# B&R Automation Studio project 305841_E00002_AM_0 (part 3)

#### GAMath.fun - Exported functions and function blocks
```iecst
(********************************************************************
 * COPYRIGHT -- General Atomics
 ********************************************************************
 * Library: GAMath
 * File: GAMathj.fun
 * Author: J Sheeron
 ********************************************************************
 * Functions and function blocks of library GAMath
 ********************************************************************)

FUNCTION_BLOCK fbCalcTrapMoveTime
  VAR_INPUT
    _I_Vel0 : REAL := 0.0; (* units/sec starting velocity *)
    _I_VelMove : REAL; (* units/sec desired move velocity*)
    _I_Accel : REAL; (* untis/sec^2 *)
    _I_Decel : REAL; (* untis/sec^2 *)
    _I_Dist : LREAL; (* units, LREAL to be compatible with motion system *)
  END_VAR

  VAR_OUTPUT
    _O_MoveTime : TIME; (* how long will the move take as a TIME type *)
    _O_MoveTimeMsec : DINT; (* mSec, how long the move will take *)
    _O_VelReached : REAL; (* units/sec. Velocity reached will be <= VelMove for triangular profiles, dist < Dcheck *)
    _O_Dcheck : LREAL; (* units. Distances > than this have a trapazoidal shape and VelReached = VelMove *)
  END_VAR

  VAR
    v0 : REAL; (* internal copy of input *)
    vMove : REAL; (* internal copy of input *)
    accel : REAL; (* internal copy of input *)
    decel : REAL; (* internal copy of input *)
    dist : LREAL; (* internal copy of input *)
    tval1  : LREAL; (* temporary value *)
    tval2  : LREAL; (* temporary value *)
    tval3  : LREAL; (* temporary value *)
    tval4  : LREAL; (* temporary value *)
    tval5  : LREAL; (* temporary value *)
    seconds : LREAL; (* temporary value *)
  END_VAR
END_FUNCTION_BLOCK

FUNCTION fctAziDiff : LREAL (* Return the angle between pos A and pos B (A-B). Returns +/- 180 deg. +: Pos A ahead of B, -: Pos A behind B *)
  (*
  Result is +/- 180 degrees
  Positive value: A is ahead of B.
  Negative value: A is behind B.
  Account for 360 deg rollover. *)
  VAR_INPUT
    _I_PosA : LREAL;
    _I_PosB : LREAL;
  END_VAR

  VAR
    angle : LREAL;
  END_VAR
END_FUNCTION

FUNCTION fctLRCeiling : LREAL (* LREAL Ceiling -- Return the smallest whole number not less than value *)
  VAR_INPUT
    _I_Val : LREAL;
  END_VAR

  VAR
    val1 : LREAL;
    rem : LREAL;
  END_VAR
END_FUNCTION

FUNCTION fctLRFloor : LREAL (* LREAL floor -- Return the largest whole number not greater than value *)
  VAR_INPUT
    _I_Val : LREAL;
  END_VAR

  VAR
    val1 : LREAL;
  END_VAR
END_FUNCTION

FUNCTION fctLRFract : LREAL (* LREAL fractional -- Return the fractional part of a value *)
  VAR_INPUT
    _I_Val : LREAL;
  END_VAR

  VAR
    val1 : LREAL;
  END_VAR
END_FUNCTION

FUNCTION fctLRMod : LREAL (* LREAL MOD -- Return the remainder of Dividend MOD Divisor *)
  VAR_INPUT
    _I_Dividend : LREAL;
    _I_Divisor : LREAL;
  END_VAR

  VAR
    val1 : LREAL;
    rem : LREAL;
  END_VAR
END_FUNCTION

FUNCTION fctRound1 : REAL (* Return the source value (real) rounded to 1 decimal place *)
  VAR_INPUT
    _I_src : LREAL; (* REAL value to be rounded *)
  END_VAR
  VAR
    dintTemp : DINT; (* temp value *)
  END_VAR
END_FUNCTION

FUNCTION fctRound2 : REAL (* Return the source value (real) rounded to 2 decimal places *)
  VAR_INPUT
    _I_src : LREAL; (* REAL value to be rounded *)
  END_VAR
  VAR
    dintTemp : DINT; (* temp value *)
  END_VAR
END_FUNCTION

FUNCTION fctRound3 : REAL (* Return the source value (real) rounded to 2 decimal places *)
  VAR_INPUT
    _I_src : LREAL; (* REAL value to be rounded *)
  END_VAR
  VAR
    dintTemp : DINT; (* temp value *)
  END_VAR
END_FUNCTION

FUNCTION fctLRound1 : LREAL (* Return the source value (LREAL) rounded to 1 decimal place *)
  VAR_INPUT
    _I_src : LREAL; (* REAL value to be rounded *)
  END_VAR
  VAR
    dintTemp : DINT; (* temp value *)
  END_VAR
END_FUNCTION

FUNCTION fctLRound2 : LREAL (* Return the source value (LREAL) rounded to 2 decimal places *)
  VAR_INPUT
    _I_src : LREAL; (* REAL value to be rounded *)
  END_VAR
  VAR
    dintTemp : DINT; (* temp value *)
  END_VAR
END_FUNCTION

FUNCTION fctLRound3 : LREAL (* Return the source value (LREAL) rounded to 2 decimal places *)
  VAR_INPUT
    _I_src : LREAL; (* REAL value to be rounded *)
  END_VAR
  VAR
    dintTemp : DINT; (* temp value *)
  END_VAR
END_FUNCTION
```

#### GAMath.st - Implementation code
```iecst
(********************************************************************
 * COPYRIGHT -- General Atomics
 ********************************************************************
 * Library: GAMath
 * File: GAMathj.st
 * Author: J Sheeron
 ********************************************************************
 * Functions and function blocks of library GAMath
 ********************************************************************)
// Estimate time needed to make a trapazoidal move
FUNCTION_BLOCK fbCalcTrapMoveTime

  // Useful motion formulas:
  //    V^2 = V0^2 + (2 * acc * dist)  OR  dist = (V^2 - V0^2) / 2acc (1)
  //    V = V0 + (acc * t)  OR  t = (V - V0) / acc                    (2)
  //    Dist = (V0*t) + (1/2 * acc * t^2)                             (3)

  // **** First, return zeros on invalid inputs.
  // Assume distance, and accel and decel cannot be zero.
  // Assume V - V0 cannot be zero
  IF _I_VelMove = 0.0 OR (_I_VelMove = _I_Vel0) OR _I_Accel = 0.0 OR _I_Decel = 0.0 OR _I_Dist = 0.0 THEN
    _O_MoveTime := T#0ms;
    _O_VelReached := 0.0;
    _O_Dcheck := 0.0;
    RETURN;
  END_IF;

  // **** Condition inputs.
  // Force accel, decel and distance to be positive.
  // Force VelMove > V0, swapping them if necessary.
  // IMPROVEMENT: Perhaps it can be made so that negative accel, decel, distance, and velocity inputs
  // are handled gracrfully. Not needed now, so leave this for later if there is time/need.
  v0 := ABS(_I_Vel0);
  vMove := ABS(_I_VelMove);
  // swap V0 and VMove if needed such that v0 < vMove
  IF v0 > vMove THEN
    v0 := ABS(_I_VelMove);
    vMove := ABS(_I_Vel0);
  END_IF;
  accel := ABS(_I_Accel);
  decel := ABS(_I_Decel);
  dist := ABS(_I_Dist);

  // **** Now figure out the move profile.
  // If the requested distance is less than or equal the check distance Dcheck,
  // the move profile is a triangle, and the move velocity will not be reached,
  // or may be reached, but not sustained.

  // If the requested distance is greater than the check distance, then the
  // move profile is trapazoidal, and the velocity will flat top at the move velocity.

  // Calculate the check distance Dcheck
  tval1 := vMove**2 - v0**2;
  tval2 := tval1 / (2 * accel); // dist accel (V^2 - V0^2) / (2*accel) (1)
  tval3 := tval1 / (2 * decel); // dist decel
  _O_Dcheck := tval2 + tval3; // Return the distance check for informational purposes.

  IF dist <= _O_Dcheck THEN
    // ** Triangular profiles
    // Profile is an accel segment and decel segemnt that meet at a point (no flat top at the MOVE velocity).
    // We need to know what velocity is reached. ** The area of the triangle is the distance traveled**,
    // and we know the accel time or distance + the decel time or distance = total time or distance, but we
    // need to know how long or how far the accel or decel component is.
    // Dist = 1/2 * acc * t^2 (3) above, so distance (area) varies linearly and inversely with acc. Furthermore,
    // we know the ratio of accel to decel, so we should be able to figure out the ratio of the distances (areas).
    // Daccel = (1 / Ratio accel:decel) * Ddecel ==> Daccel = (decel/accel) * Ddecel  OR  Ddecel = (accel / decel) * Daccel  (4)
    // Dtotal = Taccel + Tdecel. Substituing in (4) ==> Dtotal = Daccel + (accel/decel) * Daccel ==>
    // Dtotal = Daccel(1 + accel/decel) OR Daccel = Dtotal / (1 + (accel / decel))
    // The area of the acceleration portion is the trialgle with a base with a length of time Tacc, and this varies with the total time
    // by the same ratio of the accel/decel because the area of the triangle varies linearly with the length of the base
    // Taccel = (1 / Ratio accel:decel) * Tdecel ==> Taccel = (decel/accel) * Tdecel OR Tdecel = (accel / decel) * Taccel    (5)
    // Ttotal = Taccel + Tdecel. Substituing in (4) ==> Ttotal = Taccel + (accel/decel) * Taccel ==>
    // Ttotal = Taccel(1 + accel/decel) OR Taccel = Ttotal / (1 + (accel / decel))
    // So putting this all together:
    // 1) Distance traveled = area of the triangle
    // 2) The length of the base of the triangle is the total time
    // 3) Aaccel = Daccel = Dtotal / (1 + (accel / decel)
    // Then it follows that:
    // 4) V = SQRT(V0^2 + (2 * accel * Daccel))             (1)
    // 5) Ttotal = ((V - V0) / accel) + ((V - V0) / decel)  (2)
    tval1 := dist / (1 + (accel / decel));  // Daccel
    _O_VelReached := SQRT(v0**2 + (2.0 * accel * tval1)); // V = SQRT(V0^2 + (2 * acc * dist))
    tval1 := _O_VelReached - v0;
    seconds :=  (tval1 / accel) + (tval1 / decel); // Move time as a float, in seconds. t = ((V - V0) / accel) + ((V - V0) / decel)
  ELSE
    // trapazoidal profiles -- profile is an accel segment a decel segemnt,
    // and a constant velocity segment in between at the move velocity.
    // Total move time is Taccel + Tconstant + Tdecel.
    // Velocity reached = move velocity.
    _O_VelReached := vMove;

    // 1) Calculate the time it takes to accelerate to Vmove
    // Taccel = (V - V0) / accel   (2)
    // 2) Calculate the distance traveled during the acceleration segment
    // Daccel = 1/2 * accel * t^2  (3)
    // 3) Similarly calcuate Tdecel and Ddecel
    // 4) Dconstant = Dmove - (Daccel + Ddecel) Total distance less distance for accel & decel
    // 5) Tconstant = Dconstant / Vmove
    // 6) Calculate Total move time: Tmove = Taccel + Tconstant + Tdecel

    // Calc accel and decel times
    tval1 := vMove - v0;
    tval2 := tval1 / accel; // Taccel = (V - V0) / accel  (2)
    tval3 := tval1 / decel; // Tdecel

    // Calc accel and decel distances
    tval4 := (v0 * tval2) + (0.5 * accel * (tval2**2)); // Daccel = V0*t + (1/2 * accel * t^2)  (3)
    tval5 := (v0 * tval3) + (0.5 * decel * (tval3**2)); // Ddecel

    // Calc constant velocity distance: Dtotal - (Daccel + Ddecel)
    tval1 := dist - (tval4 + tval5); // Dconstant

    // Calc constant velocity time: Tconstant = Dconstant / VMove
    tval4 := tval1 / vMove; // Tconstant

    // Calc Total seconds = Tmove = Taccel + Tconstant + Tdecel
    seconds := tval2 + tval4 + tval3;
  END_IF;

  // Time calculations is:
  // 1) Converted from seconds to mSec (conversion to time expects mSecs)
  // 2) Converted from LREAL to DINT, and then returned for convenience
  // 3) Converted to a TIME and returned.
  _O_MoveTimeMsec := LREAL_TO_DINT(1000 * seconds);
  _O_MoveTime := DINT_TO_TIME(_O_MoveTimeMsec);
END_FUNCTION_BLOCK

// Return the angle between pos A and pos B (A-B). Returns +/- 180 deg. +: Pos A ahead of B, -: Pos A behind B
FUNCTION fctAziDiff
  // Positive value: A is ahead of B,
  // Negative value: A is behind B.
  // Accounts for 360 degree rollover

  angle := _I_PosA - _I_PosB;
  // Deal with 360 deg rollover and normalize result to +/- 180 deg
  // Subtract target from position.
  // If the result < -180, add 360.
  // If the result > 180, subtract 360.
  IF angle < -180.0 THEN
    angle:= angle + 360.0;
  ELSIF angle > 180.0THEN
    angle := angle - 360.0;
  END_IF;
  fctAziDiff := angle;
END_FUNCTION

// LREAL Ceiling -- Return the smallest whole number not less than value
FUNCTION fctLRCeiling
  val1 := TRUNC(_I_Val);
  rem := _I_Val - val1; // the remainder portion
  IF rem > 0 THEN
    // non-zero remainder. Round up
    fctLRCeiling := val1 + 1.0;
  ELSE
    // no remainder -- must already be a whole number
    fctLRCeiling := val1;
  END_IF;
END_FUNCTION

// LREAL Floor -- Return the largest whole number as a LREAL not greater than value
FUNCTION fctLRFloor
  val1 := TRUNC(_I_Val);  // Trunc returns an integer, but it is put into a LREAL
  fctLRFloor := val1;
END_FUNCTION

// LREAL Fract -- Return the fractional part of a value
FUNCTION fctLRFract
  val1 := TRUNC(_I_Val);
  fctLRFract := _I_Val - val1; // the remainder portion
END_FUNCTION

// MOD LREAL Return the remainder of Dividend MOD Divisor
FUNCTION fctLRMod
  val1 := _I_Dividend / _I_Divisor;
  rem := val1 - TRUNC(val1); // the remainder portion
  fctLRMod := rem * _I_Divisor; // remainder * divisor = mod
END_FUNCTION

// Return the source value (real) rounded to 1 decimal place
FUNCTION fctRound1
  dintTemp:= LREAL_TO_DINT(_I_src * 10.0);
  fctRound1:= DINT_TO_REAL(dintTemp) / 10.0;
END_FUNCTION

// Return the source value (real) rounded to 2 decimal places
FUNCTION fctRound2
  // On SG4 systems the REAL_TO_DINT function rounds.
  // Beware that on SG3 systems, it truncates.
  dintTemp:= LREAL_TO_DINT(_I_src * 100.0);
  fctRound2:= DINT_TO_REAL(dintTemp) / 100.0;
END_FUNCTION

// Return the source value (real) rounded to 3 decimal places
FUNCTION fctRound3
  // On SG4 systems the REAL_TO_DINT function rounds.
  // Beware that on SG3 systems, it truncates.
  dintTemp:= LREAL_TO_DINT(_I_src * 1000.0);
  fctRound3:= DINT_TO_REAL(dintTemp) / 1000.0;
END_FUNCTION

// Return the source value (LREAL) rounded to 1 decimal place
FUNCTION fctLRound1
  dintTemp:= LREAL_TO_DINT(_I_src * 10.0);
  fctLRound1:= DINT_TO_LREAL(dintTemp) / 10.0;
END_FUNCTION

// Return the source value (LREAL) rounded to 2 decimal places
FUNCTION fctLRound2
  // On SG4 systems the REAL_TO_DINT function rounds.
  // Beware that on SG3 systems, it truncates.
  dintTemp:= LREAL_TO_DINT(_I_src * 100.0);
  fctLRound2:= DINT_TO_LREAL(dintTemp) / 100.0;
END_FUNCTION

// Return the source value (LREAL) rounded to 3 decimal places
FUNCTION fctLRound3
  // On SG4 systems the REAL_TO_DINT function rounds.
  // Beware that on SG3 systems, it truncates.
  dintTemp:= LREAL_TO_DINT(_I_src * 1000.0);
  fctLRound3:= DINT_TO_LREAL(dintTemp) / 1000.0;
END_FUNCTION
```

### Logic.typ
```iecst
TYPE
  eAXIS_DESIGNATION :
    ( (* Physical Axes *)
    AD_UNKNOWN := 0,
    AD_SPINDLE := 1,
    AD_OUTER_ECCENTRIC := 2,
    AD_INNER_ECCENTRIC := 3,
    AD_Z := 4,
    (* Other axes *)
    AD_X := 5, (* depth *)
    AD_Y := 6, (* used ? *)
    (* virtual axis *)
    AD_HANDWHEEL := 7,
    (* VFD axis *)
    AD_CF_VFD := 8
  ) := AD_UNKNOWN;

  (* Machine specific HMI axis requests. Intended to have one of these structures per axis. *)
  sHmiAxisReqs : STRUCT
    (* Boolean requests in this section. *)
    (* (none *)
    (* numerical requests *)
    (* (none *)
    (* hmi move type and direction selection related *)
    absMoveEnable : BOOL := TRUE; (* allow move type selection by default *)
    relMoveEnable : BOOL := TRUE;
    velMoveEnable : BOOL := TRUE;
    directionPosEnable : BOOL := TRUE; (* allow direction selection by default *)
    directionNegEnable : BOOL := TRUE;
    directionShortestEnable : BOOL := TRUE;
    moveDistanceEnable : BOOL := TRUE; (* enable params by default *)
    movePositionEnable : BOOL := TRUE;
    gearInEnable : BOOL := FALSE; (* coodinated axis gear in enabled *)
    shiftEnable : BOOL := FALSE; (* coordinated axis gear offset or phase shift  enabled *)
    camInEnable : BOOL := FALSE; (* coordinated axis cam in enabled *)
    disengageEnable : BOOL := FALSE; (* coordinated axis cam in enabled *)
    moveDesignation: DINT := -1; (* per hmi. 0: Abs, 1: Rel, 2:Vel or Jog, -1 is no selection. See fctDecodeHmiMoveType *)
    direction: DINT := -1; (* per hmi. 0: pos, 1: neg, 2: shortest, -1 is no selection. See fctDecodeHmiDirection *)
    (* axis designation. Two different data types for convenience. *)
    axisNo : USINT := 0; (* default to initial so setting a value can be detected. USINT for easy use in loops *)
    axisDesignation : eAXIS_DESIGNATION := AD_UNKNOWN; (* default to initial so setting a value can be detected *)
  END_STRUCT;

  (* Machine specific HMI process requests. Intended to have one of these per machine or otherwise as needed, but not per axis. *)
  sHmiProcessReqs : STRUCT
    (* Boolean requests in this section. *)
    (* NOTE/CAUTION These request bits may get cleared/copied by memcpy/memclr
    So be careful about adding boolean requests outside of this section.
    See ClearManualReqs action for example, in OmSaveDev program.
    Bool requests above StartOfClearedRequests won't get auto cleared *)
    StartOfClearedRequests : BOOL := FALSE;
    reqAxesReset : BOOL := FALSE;
    cfReqRun : BOOL := FALSE;
    cfReqStop : BOOL := FALSE; (* NOTE: Stop triggers SM Halt directly. This allows stopping from the HMI even in the wrong mode *)
    zReqMoveUpLimit : BOOL := FALSE;
    zReqMoveDownLimit : BOOL := FALSE;
    zReqMoveLUnL : BOOL := FALSE;
    zReqMoveSoc : BOOL := FALSE;
    zReqMoveIndexUp : BOOL := FALSE;
    zReqMoveIndexDown : BOOL := FALSE;
    zReqPosSocUseCurrent : BOOL := FALSE; (* set SOC to use the current position *)
    zReqPosSocUseSpecified :  BOOL := FALSE; (* set SOC to use the specified position *)
    zReqPosLUnLUseCurrent : BOOL := FALSE; (* set load/unload to use the current position *)
    zReqPosLUnLUseSpecified :  BOOL := FALSE; (* set load/unload to use the specified position *)
    cuttingHeadMoveReqRetract : BOOL := FALSE;
    EndOfClearedRequests : BOOL := FALSE;
    (* NOTE/CAUTION Bool requests below EndOfClearedRequests won't get auto cleared *)
    camReqCalcTable : BOOL := FALSE; (* calculate a new cam table. Don't auto clear since multiple processes may use this. *)
    cfIsInPressureControl : BOOL := FALSE; (* H: Pressure ctrl, L: Speed Control *)
    cfRunEnable : BOOL := FALSE; (* enable hmi request PB *)
    zMoveUpReqEnable : BOOL := FALSE; (* enable hmi request PBs *)
    zMoveDownReqEnable : BOOL := FALSE; (* enable hmi request PBs *)
    zMoveToSocReqEnable : BOOL := FALSE; (* enable hmi request PBs *)
    zMoveToLUnLReqEnable : BOOL := FALSE; (* enable hmi request PBs *)
    (* numerical values used with requests *)
    cuttingHeadReqDepth : LREAL := 0.0;
    cfRpmCmd : REAL;
    cfPsiCmd : REAL;
    zReqPosSoc : LREAL;
    zReqPosLUnL : LREAL;
  END_STRUCT;

  (* cutting fluid vfd params is defined globally so multiple programs can have scope *)
  sCuttingFluidVfd : 	STRUCT
    isModuleOk : BOOL; (* H: interface is seen on the I/O network *)
    isAllowedToStart : BOOL; (* H: Allow to start *)
    isAllowedToRun : BOOL; (* H: Allow to run, L: Shutdown *)
    isLocated : BOOL; (* H: tank is located *)
    isRunning : BOOL; (* H: Drive is enabled *)
    isFlowEstablished : BOOL; (* H: Flow is detected *)
    isAlmLoFlow : BOOL; (* Lo flow shutdown *)
    isWarnLoFlow : BOOL; (* Lo flow warning *)
    isAlmLoLvlSw : BOOL; (* L: low level swtich in alarm *)
    isAlmLoFluid : BOOL; (* Lo Lo fluid level shutdown *)
    isWarnLoFluid : BOOL; (* Lo fluid level warning *)
    isAlmLoOutletPressure : BOOL; (* Lo Lo outlet pressure shutdown *)
    isWarnLoOutletPressure : BOOL; (* Lo outlet pressure warning *)
    isAlmHiOutletPressure : BOOL; (* Hi outlet pressure shutdown *)
    isWarnHiOutletPressure : BOOL; (* Hi outlet pressure warning *)
    isWarnLoFilterDp : BOOL;
    isWarnHiFilterDp : BOOL;
    isAlmSummary : BOOL; (* one of the below alarms is active *)
    isWarnSummary : BOOL; (* one of the below alarms is active *)
    StdStatus : UINT; (* DS402 standardized status *)
    DevSpecStatus : UINT; (* device specific status *)
    StdError : UINT; (* DS402 standardized error code *)
    DevSpecError : UINT; (* device specific error code *)
    VelCommanded : INT; (* speed ref rpm after ramp *)
    VelAct : INT; (* speed actual rpm *)
  END_STRUCT;

  sCyclePermissives : STRUCT
    isOmOk : BOOL; (* operating mode is okay *)
    isCfRdy : BOOL;
    isCfFlowEstablished : BOOL;
    allowCycleStart : BOOL; (* H: cycle start is allowed *)
    allowCycleRun : BOOL; (* H: Allow Run, L: Cycle Stop. Maintain high to allow cycle to run *)
  END_STRUCT;

  sOperatingMode : 	STRUCT
    (* requests *)
    ReqEmoReset : BOOL := FALSE;
    HmiReqCycleStart : BOOL := FALSE;
    HmiReqCycleStop : BOOL := FALSE;
    ReqCycleStart : BOOL := FALSE; (* pb or hmi *)
    ReqCycleStop : BOOL := FALSE; (* pb or hmi *)
    isInCycle : BOOL := FALSE; (* cycle has started and is running *)
    isInCycleHold : BOOL := FALSE; (* in cycle, but stopped at a hold point *)
    isStopping : BOOL := FALSE; (* cycle has started, but is being stopped *)
    (* cycle cfg *)
    ShutOffCfBeforeUnload : BOOL; (* turn off cutting fluid before going to unload pos *)
    SingleCycleInclZIndex : BOOL; (* include Z index at end of single cycle cut *)
    CycleZInPlace : BOOL; (* allow cycle *)
    HmiSubMode : SINT; (* hmi selections of submode *)
    (* mode request are in a word to allow masking and easy clearing *)
    ModeReqBits : WORD := 16#0; (* see OM_xxx constants for bit *)
    SecurityLevel : WORD := SL_UNKNOWN;
    OperatingMode : WORD := OM_UNKNOWN;
    SubMode       : WORD := OM_UNKNOWN; (* see OM_xxx_SM sub mode constants *)
    SeqStep : DINT; (* TODO: Make this an enum *)
  END_STRUCT;

  sPendant : 	STRUCT
    enableSwActive : BOOL; (* H:Allow motion *)
    enableSwWiringOk : BOOL; (* H:Ok *)
    pendantAllowMoves : BOOL; (* From safety controller. H:Allow moves *)
    emoAcivated : BOOL; (* From safety controller. H:Ok, L: EMO activated *)
    emoWiringOk : BOOL; (* From safety controller. H:Ok *)
    resetReqHandwheelCount : BOOL;
    pendantPowerOk : BOOL; (* 24 VDC button/LED power *)
    encoderPowerOk : BOOL; (* 5 VDC encoder power *)
    PBInputs : ARRAY[1..9] OF BOOL; (* Raw digital input states. Elements/Bits 1-9 correspond to PB 1-9 *)
    PBStates : ARRAY[1..9] OF BOOL; (* Push Button states. Conditioned with behavior. Elements/Bits 1-9 correspond to PB 1-9 *)
    PLCmds : ARRAY[1..9] OF BOOL; (* Pilot light cmds. Elements/Bits 1-9 correspond to PB 1-9 *)
    AxisSelectInputs : ARRAY[1..3] OF BOOL; (* Raw axis select switch inputs *)
    SpeedSelectInputs : ARRAY[1..3] OF BOOL; (* Raw speed select inputs *)
    AxisSelection : eAXIS_DESIGNATION;
    SpeedSelection : REAL;
    HandwheelCounter : DINT;
    Position : REAL;
    PositionSnapshot : REAL; (* used by process to capture a position *)
    GearRatioNumerator : DINT := 100; (* gear factor of the slave / measurment resolution of the slave *)
    GearRatioDenominator : DINT := 100; (* gear factor of the master / measurment resolution of the master *)
    tmrCountResetPulse : TP;
    fbPBs : ARRAY[1..9] OF fbProcPB;
  END_STRUCT;

END_TYPE
```

### Logic.var
```iecst
VAR CONSTANT
  (* Use constants to prevent accidental change *)
  (* axis number is per eAXIS_DESIGNATION *)
  (*
  AD_UNKNOWN := 0,
  AD_SPINDLE := 1,
  AD_OUTER_ECCENTRIC := 2,
  AD_INNER_ECCENTRIC := 3,
  AD_Z := 4,
  derrived axes
  AD_X := 5,
  AD_Y := 6,
  AD_HANDWHEEL := 7,
  AD_CF_VFD := 8
  *)
  (* Axis count is set in global so it can be used to define arrays *)
  (* AXIS_COUNT : DINT := 8; *)
  (* Set max axis velocity and accel/decel *)
  (* TODO Verify *)

  (* motor rated max *)
  (* AXIS_SPINDLE_MAX_VELOCITY : REAL := (6000.0 / 3.0) / 60.0; motor rated max, scaled into process velocity in rev/sec. 6000 rpm motor, 3:1 gearbox in rps *)
  (* process max *)
  AXIS_SPINDLE_MAX_VELOCITY : REAL := (300 / 60.0) * 3.0; (* process velocity in rev/sec. 300 rpm nominal cutting. 3x to allow up to 3x nominal *)
  AXIS_SPINDLE_MAX_ACCEL : REAL := AXIS_SPINDLE_MAX_VELOCITY / 2.0; (* get to max in 2 sec *)
  AXIS_SPINDLE_MAX_DECEL : REAL := AXIS_SPINDLE_MAX_VELOCITY * 4.0; (* allow faster stops *)
  AXIS_SPINDLE_MEAS_RESOLUTION : REAL := 0.01; (* Needs to match axis configuration view >> mappMotion setting for the axis *)

  (* motor rated max *)
  AXIS_OUTE_MAX_VELOCITY : REAL := (6000.0 / 25.0) * 360 / 60.0; (* motor max in deg/sec *)
  (* process max *)
  (* AXIS_OUTE_MAX_VELOCITY : REAL := (((4.7 * 25.4) / (50.0 * 3.14159)) * 360.0 / 60.0) * 4.0; (* process max in deg/sec. 4.7 in/min converted to deg/sec. 4x to allow up to 4x nominal *)
  AXIS_OUTE_MAX_ACCEL : REAL := AXIS_OUTE_MAX_VELOCITY / 1.0; (* get to max in 1 sec *)
  AXIS_OUTE_MAX_DECEL : REAL := AXIS_OUTE_MAX_ACCEL * 4.0; (* allow faster stops *)
  AXIS_OUTE_MEAS_RESOLUTION : REAL := 0.001; (* Needs to match axis configuration view >> mappMotion setting for the axis *)

  (* motor rated max *)
  AXIS_INE_MAX_VELOCITY : REAL := (6000.0 / 25.0) * 360 / 60.0; (* motor max in deg/sec *)
  (* AXIS_INE_MAX_VELOCITY : REAL := (((4.7 * 25.4) / (50.0 * 3.14159)) * 360.0 / 60.0) * 4.0;  process max in deg/sec. 4.7 in/min converted to deg/sec. 4x to allow up to 4x nominal *)
  AXIS_INE_MAX_ACCEL : REAL := AXIS_INE_MAX_VELOCITY / 1.0; (* get to max in 1 sec *)
  AXIS_INE_MAX_DECEL : REAL := AXIS_INE_MAX_ACCEL * 4.0; (* allow faster stops *)
  AXIS_INE_MEAS_RESOLUTION : REAL := 0.001; (* Needs to match axis configuration view >> mappMotion setting for the axis *)

  (* motor rated max *)
  (* AXIS_Z_MAX_VELOCITY : REAL := (3000.0 / 60.0) * 5.0; 3000 rpm motor, 5:1 lead, mm/sec *)
  (* limit due to need for mech adjustment *)
  AXIS_Z_MAX_VELOCITY : REAL := 50.0;
  AXIS_Z_MAX_ACCEL : REAL := AXIS_Z_MAX_VELOCITY / 2.0;
  AXIS_Z_MAX_DECEL : REAL := AXIS_Z_MAX_VELOCITY * 4.0; (* allow faster stops *)
  AXIS_Z_MEAS_RESOLUTION : REAL := 0.001; (* Needs to match axis configuration view >> mappMotion setting for the axis *)

  AXIS_HW_MEAS_RESOLUTION : REAL := 0.01; (* Needs to match axis configuration view >> mappMotion setting for the axis *)

  AXIS_CFVFD_MAX_VELOCITY : REAL := 1175.0 / 60.0; (* RPS *)
  AXIS_CFVFD_MAX_ACCEL : REAL := AXIS_CFVFD_MAX_VELOCITY; (* to max in 1 sec *)
  AXIS_CFVFD_MAX_DECEL : REAL := AXIS_CFVFD_MAX_VELOCITY; (* from max in 1 sec *)

  (* Operating Mode *)
  (* in increasing order of automation no motion -> manual -> production *)
  (* requests are bit packed, so pick values for easy masking *)
  (* Use constants instead of enum so word/bit operations are legal *)
  OM_UNKNOWN : WORD             := 16#00;  (* all bits clear *)
  OM_INITIAL : WORD             := 16#01;  (* bit 0 *)
  OM_SAFE_MODE : WORD           := 16#02;  (* bit 1 *)
  OM_EMO_MODE : WORD            := 16#04;  (* bit 2 *)
  OM_CHECK_MODE : WORD          := 16#08;  (* bit 3 *)
  OM_MANUAL_MODE : WORD         := 16#10;  (* bit 4 *)
  OM_PENDANT_MODE : WORD        := 16#20;  (* bit 5 *)
  OM_PRODUCTION_MODE : WORD     := 16#40;  (* bit 6 *)
  (* sub modes *)
  OM_PROD_SM_CONTINUOUS : WORD  := 16#40; (* bit 6. Run a continuous (normal) cycle *)
  OM_PROD_SM_SINGLE : WORD      := 16#41; (* bits 6, 0. Run a single cycle *)
  OM_PROD_SM_STEPPED : WORD     := 16#42; (* bits 6, 1. Run a stepped cycle *)

  (* Security Level *)
  (* values should be in increasing levels of permsision *)
  (* Anything above 1 should have some operating permission -- i.e. can leave safe mode *)
  (* chose bits to allow easy masking and combinations *)
  (* Use constants instead of enum so word/bit operations are legal *)
  SL_UNKNOWN : WORD        := 16#0;  (* all bits clear *)
  SL_GUEST : WORD          := 16#1;  (* bit 0 *)
  SL_OPERATOR : WORD       := 16#2;  (* bit 1 *)
  SL_SUPERVISOR : WORD     := 16#4;  (* bit 2 *)
  SL_ENGINEER : WORD       := 16#8;  (* bit 3 *)
  SL_SUPERUSER : WORD      := 16#10; (* bit 4 *)

  (* process tolerances *)
  TOL_DEPTH_ZERO_DEG : LREAL := 0.002; (* degrees. Values less than this are considered zero. LREAL to be comparable to positions. TODO: Need proper value *)
  TOL_ZINDEX  : LREAL := 0.1; (* Somewhat arbitrarily of 0.1mm TODO: determine proper value *)

END_VAR

VAR
  blink025Hz : BOOL; (* 0.25 Hz blink *)
  blink050Hz : BOOL; (* 0.50 Hz blink *)
  blink100Hz : BOOL; (* 1.00 Hz blink *)

  (* IO Module Health *)
  ModStat_PLC_201 : sRioModuleHealth;
  ModStat_OWS_PLK1 : sRioModuleHealth;
  ModStat_JB1_PLK2 : sRioModuleHealth;

  (* array of axis structures *)
  axes : ARRAY[0..AXIS_COUNT] OF sMot_Axis; (* element 0 is used as a dummy axis -- an address to reference that is not an axis *)

  (* cutting fluid VFD *)
  cfVfd: sCuttingFluidVfd;

  (* global axis commands *)
  gMotionCommands : sMot_GlobalCommands; (*command structure for global command*)

  (* Operating Mode and security level *)
  operatingMode : sOperatingMode;

  (* cycle permissives *)
  cyclePermissives : sCyclePermissives;

  (* OWS Pendant *)
  owsPendant : sPendant;

  (* HMI process specific requests *)
  hmiProcessReqs : sHmiProcessReqs; (* process specific reqs *)

  (* analog inputs *)
	AI_FT_CFFlow : sAnalogInput;
	AI_LT_CFTankLevel : sAnalogInput;
	AI_PT_CFPumpOutlet : sAnalogInput;
  AI_PT_CFFilterOutlet : sAnalogInput;
  AI_DP_CFFilter : sAnalogInput;  (* virtual input derrived from 2 PTs *)

  (* digital inputs *)
	DI_LSL_CFTank : sDigitalInput;
	DI_ZS_CFTankLocator : sDigitalInput;
  DI_JI_480VACOk : sDigitalInput;
  (* digital outputs *)
  (* pb lamps *)
  DO_PB_OWSGreen : BOOL;
  DO_PB_OWSRed : BOOL;
  (* pilot lights *)
  DO_PL_OWSGreen : BOOL;
  DO_PL_OWSAmber : BOOL;
  DO_PL_OWSRed : BOOL;
  (* becon *)
  DO_PL_OWSBeconRed : BOOL;
	DO_PL_OWSBeconAmber : BOOL;
  DO_PL_OWSBeconGreen : BOOL;

END_VAR
```

### Program Logical/PlcLogic/ProcInputs (IEC)

#### ProcInputs.var - Local variables
```iecst
VAR RETAIN

END_VAR

VAR CONSTANT
  TURCK_PS5XX_100_GRADIENT : LREAL := 0.0018084817795460700;
  TURCK_PS5XX_100_OFFSET : LREAL   := -9.2594267112758800;
END_VAR

VAR
  (* set default values -- not normally needed due to global
  permanent retained status of parameters, but use for special
  cases like first startup after major change, etc. *)
  reqSetDefaultValues : BOOL := FALSE;

  (* analog scale and alarm fbs *)
  fbAI_FT_CFFlow : fbSclAlmAI;
  fbAI_LT_CFTankLevel : fbSclAlmAI;
  fbAI_PT_CFPumpOutlet : fbSclAlmAI;
  fbAI_PT_CFFilterOutlet : fbSclAlmAI;
  fbAI_DP_CFFilter : fbSclAlmAI; (* virtual input derrived from 2 PTs *)

  (* externally mapped and calculated values for Turck IO-Link pressure sensors *)
  AI_PT_CFPumpOutletRaw : UINT;
  AI_PT_CFFilterOutletRaw : UINT;

  (* digital inputs *)
  fbDI_LSL_CFTank : fbProcDI;
  fbDI_ZS_CFTankLocator : fbProcDI;
  fbDI_JI_480VACOk : fbProcDI;

END_VAR
```

#### ProcInputs.st - Cyclic code
```iecst
PROGRAM _INIT

  // **** INIT Input Processing
  // Init function blocks
  // Set the reference to the input strucures,
  // set the sentinel value, and init the fb
  // Set the channel health for the sensor to OK if the module type used does not report channel health

  // ** Analog Inputs

  // ** Cutting Fluid Pump Flow Transmitter
  // NOTE: No sensor initially fitted -- here for future use
  fbAI_FT_CFFlow._InInputStruct:= ADR(AI_FT_CFFlow);
  fbAI_FT_CFFlow._InParamsStruct := ADR(gr_AI_FT_CFFlow_Params);
  fbAI_FT_CFFlow._InSentinel:= INVALID_SENTINEL_REAL;
  fbAI_FT_CFFlow(_InSetParams:= TRUE);
  fbAI_FT_CFFlow._InSetParams:= FALSE;

  // ** Cutting Fluid Tank Level Transmitter
  // NOTE: No sensor initially fitted -- here for future use
  fbAI_LT_CFTankLevel._InInputStruct:= ADR(AI_LT_CFTankLevel);
  fbAI_LT_CFTankLevel._InParamsStruct := ADR(gr_AI_LT_CFTankLevel_Params);
  fbAI_LT_CFTankLevel._InSentinel:= INVALID_SENTINEL_REAL;
  fbAI_LT_CFTankLevel(_InSetParams:= TRUE);
  fbAI_LT_CFTankLevel._InSetParams:= FALSE;

  // ** Cutting Fluid Filter Outlet Pressure Transmitter
  fbAI_PT_CFFilterOutlet._InInputStruct:= ADR(AI_PT_CFFilterOutlet);
  fbAI_PT_CFFilterOutlet._InParamsStruct := ADR(gr_AI_PT_CFFilterOutlet_Params);
  fbAI_PT_CFFilterOutlet._InSentinel:= INVALID_SENTINEL_REAL;
  fbAI_PT_CFFilterOutlet(_InSetParams:= TRUE);
  fbAI_PT_CFFilterOutlet._InSetParams:= FALSE;

  // ** Cutting Fluid Pump Outlet Pressure Transmitter
  fbAI_PT_CFPumpOutlet._InInputStruct:= ADR(AI_PT_CFPumpOutlet);
  fbAI_PT_CFPumpOutlet._InParamsStruct := ADR(gr_AI_PT_CFPumpOutlet_Params);
  fbAI_PT_CFPumpOutlet._InSentinel:= INVALID_SENTINEL_REAL;
  fbAI_PT_CFPumpOutlet(_InSetParams:= TRUE);
  fbAI_PT_CFPumpOutlet._InSetParams:= FALSE;

  // ** Cutting Fluid Pump Filter Differential Pressure Transmitter
  // Note: This is a 'virtual' instrument -- the dp across the filter is derrived
  // from the two pressure transducers. Use the Real input type -- it does not need scaling,
  // but does need alarming.
  gr_AI_DP_CFFilter_Params.RawType := GAPIO_RWST_REAL;
  fbAI_DP_CFFilter._InInputStruct:= ADR(AI_DP_CFFilter);
  fbAI_DP_CFFilter._InParamsStruct := ADR(gr_AI_DP_CFFilter_Params);
  fbAI_DP_CFFilter._InSentinel:= INVALID_SENTINEL_REAL;
  fbAI_DP_CFFilter(_InSetParams:= TRUE);
  fbAI_DP_CFFilter._InSetParams:= FALSE;

  // ** Digital Inputs
  fbDI_JI_480VACOk._InInputStruct:= ADR(DI_JI_480VACOk);
  fbDI_JI_480VACOk._InParamsStruct:= ADR(gr_DI_JI_480VACOk_Params);
  fbDI_JI_480VACOk._InSentinel:= FALSE;
  fbDI_JI_480VACOk(_InSetParams:= TRUE);
  fbDI_JI_480VACOk._InSetParams:= FALSE;

  fbDI_LSL_CFTank._InInputStruct:= ADR(DI_LSL_CFTank);
  fbDI_LSL_CFTank._InParamsStruct:= ADR(gr_DI_LSL_CFTank_Params);
  fbDI_LSL_CFTank._InSentinel:= FALSE;
  fbDI_LSL_CFTank(_InSetParams:= TRUE);
  fbDI_LSL_CFTank._InSetParams:= FALSE;

  fbDI_ZS_CFTankLocator._InInputStruct:= ADR(DI_ZS_CFTankLocator);
  fbDI_ZS_CFTankLocator._InParamsStruct:= ADR(gr_DI_ZS_CFTankLocator_Params);
  fbDI_ZS_CFTankLocator._InSentinel:= FALSE;
  fbDI_ZS_CFTankLocator(_InSetParams:= TRUE);
  fbDI_ZS_CFTankLocator._InSetParams:= FALSE;
END_PROGRAM

PROGRAM _CYCLIC

  // Set the default params on request, and then clear the request.
  // NOTE: This is not normally needed due to global
  // permanent retained status of parameters, but use for special
  // cases like first startup after major change, or to make sure
  // values are set to known, observable values.
  IF reqSetDefaultValues THEN
    SetInputParams;
    reqSetDefaultValues := FALSE;
  END_IF;

  // **** Run the analog and digital input processing
  // The input signals are generally mapped in the I/O mapping, unless there is a
  // further conditioning or logic needed.
  // Map the ModuleOk, ChannelOk, and run the fb.
  // If the channel OK is not available in the hardware I/O mapping,
  // either do it manually, or use the Module OK for the channel ok.

  // ** Analog Inputs

  AI_FT_CFFlow.ModuleOk:= ModStat_JB1_PLK2.Slot04ModuleOk;
  fbAI_FT_CFFlow();

  AI_LT_CFTankLevel.ModuleOk:= ModStat_JB1_PLK2.Slot04ModuleOk;
  fbAI_LT_CFTankLevel();

  AI_PT_CFPumpOutlet.ModuleOk:= ModStat_JB1_PLK2.Slot05ModuleOk;
  AI_PT_CFPumpOutlet.ChannelOk := AI_PT_CFPumpOutlet.ModuleOk; // TODO: Update. Need to figure out what is needed in the IO-Link case.
  // Manually set the raw input, externally calc scaling, and then call the fb.
  // Mfg formula gives pressure in bar, and then convert to psig.
  AI_PT_CFPumpOutlet.InRawUINT := AI_PT_CFPumpOutletRaw;
  AI_PT_CFPumpOutlet.InScaled := LREAL_TO_REAL(((UINT_TO_LREAL(AI_PT_CFPumpOutletRaw) * TURCK_PS5XX_100_GRADIENT) + TURCK_PS5XX_100_OFFSET) * 14.50377);
  fbAI_PT_CFPumpOutlet();

  AI_PT_CFFilterOutlet.ModuleOk:= ModStat_JB1_PLK2.Slot05ModuleOk;
  AI_PT_CFFilterOutlet.ChannelOk := AI_PT_CFFilterOutlet.ModuleOk; // TODO: Update. Need to figure out what is needed in the IO-Link case.
  // Manually set the raw input, externally calc scaling, and then call the fb.
  // Mfg formula gives pressure in bar, and then convert to psig.
  AI_PT_CFFilterOutlet.InRawUINT := AI_PT_CFFilterOutletRaw;
  AI_PT_CFFilterOutlet.InScaled := LREAL_TO_REAL(((UINT_TO_LREAL(AI_PT_CFFilterOutletRaw) * TURCK_PS5XX_100_GRADIENT) + TURCK_PS5XX_100_OFFSET) * 14.50377);
  fbAI_PT_CFFilterOutlet();

  // The 'virtual' CF Filter DP is derrived from two real PTs across the filter/
  // And the module and channel okays. Subtract the PVs to get the new signal.
  AI_DP_CFFilter.ModuleOk:= AI_PT_CFPumpOutlet.ModuleOk AND AI_PT_CFFilterOutlet.ModuleOk;
  AI_DP_CFFilter.ChannelOk := AI_PT_CFPumpOutlet.ChannelOk AND AI_PT_CFFilterOutlet.ChannelOk;
  AI_DP_CFFilter.InRawREAL := AI_PT_CFPumpOutlet.InScaledFiltered - AI_PT_CFFilterOutlet.InScaledFiltered;
  fbAI_DP_CFFilter();

  // ** Digital Inputs
  DI_JI_480VACOk.ModuleOk := ModStat_PLC_201.Slot01ModuleOk;
  DI_JI_480VACOk.ChannelOk := DI_JI_480VACOk.ModuleOk;
  fbDI_JI_480VACOk();

  DI_LSL_CFTank.ModuleOk := ModStat_JB1_PLK2.Slot02ModuleOk;
  DI_LSL_CFTank.ChannelOk := DI_LSL_CFTank.ModuleOk;
  fbDI_LSL_CFTank();

  DI_ZS_CFTankLocator.ModuleOk := ModStat_JB1_PLK2.Slot02ModuleOk;
  DI_ZS_CFTankLocator.ChannelOk := DI_ZS_CFTankLocator.ModuleOk;
  fbDI_ZS_CFTankLocator;

END_PROGRAM

PROGRAM _EXIT
	(* Insert code here *)

END_PROGRAM
```

#### Action.st
```iecst
ACTION SetInputParams:
  // Default CF Flow Params
  gr_AI_FT_CFFlow_Params.LpEnable := FALSE;
  gr_AI_FT_CFFlow_Params.LpPreserveUnfiltered := TRUE; //F: unfiltered = filtered, T: keep separate
  gr_AI_FT_CFFlow_Params.AlmEnable := FALSE; // Not fitted. Set once fitted to enable alarming
  gr_AI_FT_CFFlow_Params.AlmLoLoEnable := TRUE;
  gr_AI_FT_CFFlow_Params.AlmLoEnable := TRUE;
  gr_AI_FT_CFFlow_Params.AlmHiEnable := FALSE;
  gr_AI_FT_CFFlow_Params.AlmHiHiEnable := FALSE; // alarm thresholds - compare to EU (scaled) values
  gr_AI_FT_CFFlow_Params.RawType := GAPIO_RWST_INT;
  // scaling parameters
  // scaling TBD
  gr_AI_FT_CFFlow_Params.CalcEUExternally := FALSE;
  gr_AI_FT_CFFlow_Params.RawMin := 0.0;
  gr_AI_FT_CFFlow_Params.RawMax := 32767.0;
  gr_AI_FT_CFFlow_Params.EuMin := 0.0;
  gr_AI_FT_CFFlow_Params.EuMax := 100.0;
  gr_AI_FT_CFFlow_Params.RawOffset := 0.0; // +/- counts value added to the raw value before scaling
  gr_AI_FT_CFFlow_Params.EuOffset := 0.0; // +/- EU value added to EU after scaling
  // Low Pass (Noise) filter parameters
  gr_AI_FT_CFFlow_Params.LpCoeff := 0.0; // >=0 and <1. 0= no filtering. 0.99999= heavy filtering.
  // alarm enables
  gr_AI_FT_CFFlow_Params.AlmRangeThreshLo := -1.0E9;
  gr_AI_FT_CFFlow_Params.AlmRangeThreshHi := 1.0E9;
  gr_AI_FT_CFFlow_Params.AlmThreshLoLo := -1.0E9;
  gr_AI_FT_CFFlow_Params.AlmThreshLo := -1.0E9;
  gr_AI_FT_CFFlow_Params.AlmThreshHi := 1.0E9;
  gr_AI_FT_CFFlow_Params.AlmThreshHiHi := 1.0E9;
  // Alarm deadbands in % of range EU range. Use 0.0 to disable
  gr_AI_FT_CFFlow_Params.AlmDbLoPct := 1.0; // pvs must rise above threshold by the corresponding value in order to be considered clear
  gr_AI_FT_CFFlow_Params.AlmDbHiPct := 1.0; // pvs must drop below threshold by the corresponding value in order to be considered clear
  // alarm time delays. Use T#0ms time to disable
  gr_AI_FT_CFFlow_Params.AlmLoOnDlyTime := T#5s;
  gr_AI_FT_CFFlow_Params.AlmHiOnDlyTime := T#1s;
  // alarm off delay time - condition must clear for this long before being considered "gone"
  gr_AI_FT_CFFlow_Params.AlmLoOffDlyTime := T#1s;
  gr_AI_FT_CFFlow_Params.AlmHiOffDlyTime := T#1s;

  // Default Tank Level Params
  gr_AI_LT_CFTankLevel_Params.LpEnable := FALSE;
  gr_AI_LT_CFTankLevel_Params.LpPreserveUnfiltered := TRUE; //F: unfiltered = filtered, T: keep separate
  gr_AI_LT_CFTankLevel_Params.AlmEnable := FALSE; // Not fitted. Set once fitted to enable alarming
  gr_AI_LT_CFTankLevel_Params.AlmLoLoEnable := TRUE;
  gr_AI_LT_CFTankLevel_Params.AlmLoEnable := TRUE;
  gr_AI_LT_CFTankLevel_Params.AlmHiEnable := FALSE;
  gr_AI_LT_CFTankLevel_Params.AlmHiHiEnable := FALSE; // alarm thresholds - compare to EU (scaled) values
  gr_AI_LT_CFTankLevel_Params.RawType := GAPIO_RWST_INT;
  // scaling parameters
  // scaling TBD
  gr_AI_LT_CFTankLevel_Params.CalcEUExternally := FALSE;
  gr_AI_LT_CFTankLevel_Params.RawMin := 0.0;
  gr_AI_LT_CFTankLevel_Params.RawMax := 32767.0;
  gr_AI_LT_CFTankLevel_Params.EuMin := 0.0;
  gr_AI_LT_CFTankLevel_Params.EuMax := 100.0;
  gr_AI_LT_CFTankLevel_Params.RawOffset := 0.0; // +/- counts value added to the raw value before scaling
  gr_AI_LT_CFTankLevel_Params.EuOffset := 0.0; // +/- EU value added to EU after scaling
  // Low Pass (Noise) filter parameters
  gr_AI_LT_CFTankLevel_Params.LpCoeff := 0.0; // >=0 and <1. 0= no filtering. 0.99999= heavy filtering.
  // alarm enables
  gr_AI_LT_CFTankLevel_Params.AlmRangeThreshLo := -1.0E9;
  gr_AI_LT_CFTankLevel_Params.AlmRangeThreshHi := 1.0E9;
  gr_AI_LT_CFTankLevel_Params.AlmThreshLoLo := -1.0E9;
  gr_AI_LT_CFTankLevel_Params.AlmThreshLo := -1.0E9;
  gr_AI_LT_CFTankLevel_Params.AlmThreshHi := 1.0E9;
  gr_AI_LT_CFTankLevel_Params.AlmThreshHiHi := 1.0E9;
  // Alarm deadbands in % of range EU range. Use 0.0 to disable
  gr_AI_LT_CFTankLevel_Params.AlmDbLoPct := 1.0; // pvs must rise above threshold by the corresponding value in order to be considered clear
  gr_AI_LT_CFTankLevel_Params.AlmDbHiPct := 1.0; // pvs must drop below threshold by the corresponding value in order to be considered clear
  // alarm time delays. Use T#0ms time to disable
  gr_AI_LT_CFTankLevel_Params.AlmLoOnDlyTime := T#5s;
  gr_AI_LT_CFTankLevel_Params.AlmHiOnDlyTime := T#1s;
  // alarm off delay time - condition must clear for this long before being considered "gone"
  gr_AI_LT_CFTankLevel_Params.AlmLoOffDlyTime := T#1s;
  gr_AI_LT_CFTankLevel_Params.AlmHiOffDlyTime := T#1s;

  // Default Pump Outlet Pressure Params
  gr_AI_PT_CFPumpOutlet_Params.LpEnable := TRUE;
  gr_AI_PT_CFPumpOutlet_Params.LpPreserveUnfiltered := TRUE; //F: unfiltered = filtered, T: keep separate
  // gr_AI_PT_CFPumpOutlet_Params.AlmEnable := TRUE; // Dynamic, set in CF VFD
  gr_AI_PT_CFPumpOutlet_Params.AlmLoLoEnable := TRUE;
  gr_AI_PT_CFPumpOutlet_Params.AlmLoEnable := TRUE;
  gr_AI_PT_CFPumpOutlet_Params.AlmHiEnable := TRUE;
  gr_AI_PT_CFPumpOutlet_Params.AlmHiHiEnable := TRUE; // alarm thresholds - compare to EU (scaled) values
  gr_AI_PT_CFPumpOutlet_Params.RawType := GAPIO_RWST_UINT; // UINT in the IO-Link case
  // scaling parameters
  // IO-Link is scaled at the device, but adheres to a mfg given formula
  // Pressure in bar = (measured value * Gradient) + Offset
  // This calc is done and the scaled value is set outside the fb
  gr_AI_PT_CFPumpOutlet_Params.CalcEUExternally := TRUE; // CALC EU Outside scaling fb!!
  gr_AI_PT_CFPumpOutlet_Params.RawMin := 5120.0;
  gr_AI_PT_CFPumpOutlet_Params.RawMax := 60415.0;
  gr_AI_PT_CFPumpOutlet_Params.EuMin := 0.0;  // 0-100 BAR in PSI but not used directly with external calc scaling
  gr_AI_PT_CFPumpOutlet_Params.EuMax := 1450.38;
  gr_AI_PT_CFPumpOutlet_Params.RawOffset := 0.0; // +/- counts value added to the raw value before scaling
  gr_AI_PT_CFPumpOutlet_Params.EuOffset := 0.0; // +/- EU value added to EU after scaling
  // Low Pass (Noise) filter parameters
  gr_AI_PT_CFPumpOutlet_Params.LpCoeff := 0.99; // >=0 and <1. 0= no filtering. 0.99999= heavy filtering.
  // alarm enables
  gr_AI_PT_CFPumpOutlet_Params.AlmRangeThreshLo := -10.0; // allow some negative pressure gr_AI_PT_CFPumpOutlet_Params.EuMin;
  gr_AI_PT_CFPumpOutlet_Params.AlmRangeThreshHi := gr_AI_PT_CFPumpOutlet_Params.EuMax;
  gr_AI_PT_CFPumpOutlet_Params.AlmThreshLoLo := 25.0; // TODO: Figure out the alm thresholds
  gr_AI_PT_CFPumpOutlet_Params.AlmThreshLo := 30.0;
  // Seal has a 300 PSI limit but be conservative at 250 -- keep 'er under this
  gr_AI_PT_CFPumpOutlet_Params.AlmThreshHi := 225.0;
  gr_AI_PT_CFPumpOutlet_Params.AlmThreshHiHi := 250.0;
  // Alarm deadbands in % of range EU range. Use 0.0 to disable
  // Specified here in EU, and converted to a percent
  gr_AI_PT_CFPumpOutlet_Params.AlmDbLoPct := (3.0 / (gr_AI_PT_CFPumpOutlet_Params.EuMax - gr_AI_PT_CFPumpOutlet_Params.EuMin)) * 100.0; // pvs must rise above threshold by the corresponding value in order to be considered clear
  gr_AI_PT_CFPumpOutlet_Params.AlmDbHiPct := (3.0 / (gr_AI_PT_CFPumpOutlet_Params.EuMax - gr_AI_PT_CFPumpOutlet_Params.EuMin)) * 100.0; // pvs must drop below threshold by the corresponding value in order to be considered clear
  // alarm time delays. Use T#0ms time to disable
  gr_AI_PT_CFPumpOutlet_Params.AlmLoOnDlyTime := T#5s;
  gr_AI_PT_CFPumpOutlet_Params.AlmHiOnDlyTime := T#5s;
  // alarm off delay time - condition must clear for this long before being considered "gone"
  gr_AI_PT_CFPumpOutlet_Params.AlmLoOffDlyTime := T#1s;
  gr_AI_PT_CFPumpOutlet_Params.AlmHiOffDlyTime := T#1s;

  // Default Filter Outlet Pressure Params
  gr_AI_PT_CFFilterOutlet_Params.LpEnable := TRUE;
  gr_AI_PT_CFFilterOutlet_Params.LpPreserveUnfiltered := TRUE; // F: unfiltered = filtered, T: keep separate
  gr_AI_PT_CFFilterOutlet_Params.AlmEnable := FALSE;
  gr_AI_PT_CFFilterOutlet_Params.AlmLoLoEnable := TRUE;
  gr_AI_PT_CFFilterOutlet_Params.AlmLoEnable := TRUE;
  gr_AI_PT_CFFilterOutlet_Params.AlmHiEnable := TRUE;
  gr_AI_PT_CFFilterOutlet_Params.AlmHiHiEnable := TRUE; // alarm thresholds - compare to EU (scaled) values
  gr_AI_PT_CFFilterOutlet_Params.RawType := GAPIO_RWST_UINT; // UINT in the IO-Link case
  // scaling parameters
  // IO-Link is scaled at the device
  gr_AI_PT_CFFilterOutlet_Params.CalcEUExternally := TRUE; // CALC EU Outside scaling fb!!
  gr_AI_PT_CFFilterOutlet_Params.RawMin := 5120.0;
  gr_AI_PT_CFFilterOutlet_Params.RawMax := 60415.0;
  gr_AI_PT_CFFilterOutlet_Params.EuMin := 0.0;  // 0-100 BAR in PSI but not used directly with external calc scaling
  gr_AI_PT_CFFilterOutlet_Params.EuMax := 1450.38;
  gr_AI_PT_CFFilterOutlet_Params.RawOffset := 0.0; // +/- counts value added to the raw value before scaling
  gr_AI_PT_CFFilterOutlet_Params.EuOffset := 0.0; // +/- EU value added to EU after scaling
  // Low Pass (Noise) filter parameters
  gr_AI_PT_CFFilterOutlet_Params.LpCoeff := 0.99; // >=0 and <1. 0= no filtering. 0.99999= heavy filtering.
  // alarm enables
  gr_AI_PT_CFFilterOutlet_Params.AlmRangeThreshLo := -10.0; // allow some negative pressure gr_AI_PT_CFFilterOutlet_Params.EuMin;
  gr_AI_PT_CFFilterOutlet_Params.AlmRangeThreshHi := gr_AI_PT_CFFilterOutlet_Params.EuMax;
  gr_AI_PT_CFFilterOutlet_Params.AlmThreshLoLo := 25.0;
  gr_AI_PT_CFFilterOutlet_Params.AlmThreshLo := 30.0;
  // Seal has a 300 PSI limit and there is some other limitation at 150 PSI-- keep 'er under this
  gr_AI_PT_CFFilterOutlet_Params.AlmThreshHi := 75.0;
  gr_AI_PT_CFFilterOutlet_Params.AlmThreshHiHi := 80.0;
  // Alarm deadbands in % of range EU range. Use 0.0 to disable
  // Specified here in EU, and converted to a percent
  gr_AI_PT_CFFilterOutlet_Params.AlmDbLoPct := (3.0 / (gr_AI_PT_CFFilterOutlet_Params.EuMax - gr_AI_PT_CFFilterOutlet_Params.EuMin)) * 100.0; // pvs must rise above threshold by the corresponding value in order to be considered clear
  gr_AI_PT_CFFilterOutlet_Params.AlmDbHiPct := (3.0 / (gr_AI_PT_CFFilterOutlet_Params.EuMax - gr_AI_PT_CFFilterOutlet_Params.EuMin)) * 100.0; // pvs must drop below threshold by the corresponding value in order to be considered clear
  // alarm time delays. Use T#0ms time to disable
  gr_AI_PT_CFFilterOutlet_Params.AlmLoOnDlyTime := T#5s;
  gr_AI_PT_CFFilterOutlet_Params.AlmHiOnDlyTime := T#5s;
  // alarm off delay time - condition must clear for this long before being considered "gone"
  gr_AI_PT_CFFilterOutlet_Params.AlmLoOffDlyTime := T#1s;
  gr_AI_PT_CFFilterOutlet_Params.AlmHiOffDlyTime := T#1s;

  // Default Filter Outlet Pressure Params
  // "Virtual" input derrived from the 2 PTs above
  gr_AI_DP_CFFilter_Params.LpEnable := TRUE;
  gr_AI_DP_CFFilter_Params.LpPreserveUnfiltered := TRUE; //F: unfiltered = filtered, T: keep separate
  // gr_AI_DP_CFFilter_Params.AlmEnable := TRUE; // Dynamic, set in CF VFD
  gr_AI_DP_CFFilter_Params.AlmLoLoEnable := FALSE;
  gr_AI_DP_CFFilter_Params.AlmLoEnable := FALSE;
  gr_AI_DP_CFFilter_Params.AlmHiEnable := TRUE;
  gr_AI_DP_CFFilter_Params.AlmHiHiEnable := TRUE; // alarm thresholds - compare to EU (scaled) values
  gr_AI_DP_CFFilter_Params.RawType := GAPIO_RWST_REAL;
  // scaling parameters
  // IO-Link is scaled at the device
  gr_AI_DP_CFFilter_Params.RawMin := -10.0; // allow for some miscalibration
  gr_AI_DP_CFFilter_Params.RawMax := 1450.38;
  gr_AI_DP_CFFilter_Params.EuMin := -10.0;
  gr_AI_DP_CFFilter_Params.EuMax := 1450.38;
  gr_AI_DP_CFFilter_Params.RawOffset := 0.0; // +/- counts value added to the raw value before scaling
  gr_AI_DP_CFFilter_Params.EuOffset := 0.0; // +/- EU value added to EU after scaling
  // Low Pass (Noise) filter parameters
  gr_AI_DP_CFFilter_Params.LpCoeff := 0.99; // >=0 and <1. 0= no filtering. 0.99999= heavy filtering.
  // alarm enables
  // TBD
  gr_AI_DP_CFFilter_Params.AlmRangeThreshLo := gr_AI_DP_CFFilter_Params.EuMin;
  gr_AI_DP_CFFilter_Params.AlmRangeThreshHi := gr_AI_DP_CFFilter_Params.EuMax;
  gr_AI_DP_CFFilter_Params.AlmThreshLoLo := gr_AI_DP_CFFilter_Params.EuMin;
  gr_AI_DP_CFFilter_Params.AlmThreshLo := gr_AI_DP_CFFilter_Params.EuMin;
  gr_AI_DP_CFFilter_Params.AlmThreshHi := 10.0;
  gr_AI_DP_CFFilter_Params.AlmThreshHiHi := 20.0;
  // Alarm deadbands in % of range EU range. Use 0.0 to disable
  // Specified here in EU, and converted to a percent
  gr_AI_DP_CFFilter_Params.AlmDbLoPct := (1.0 / (gr_AI_DP_CFFilter_Params.EuMax - gr_AI_DP_CFFilter_Params.EuMin)) * 100.0; // pvs must rise above threshold by the corresponding value in order to be considered clear
  gr_AI_DP_CFFilter_Params.AlmDbHiPct := (1.0 / (gr_AI_DP_CFFilter_Params.EuMax - gr_AI_DP_CFFilter_Params.EuMin)) * 100.0; // pvs must drop below threshold by the corresponding value in order to be considered clear
  // alarm time delays. Use T#0ms time to disable
  gr_AI_DP_CFFilter_Params.AlmLoOnDlyTime := T#5s;
  gr_AI_DP_CFFilter_Params.AlmHiOnDlyTime := T#5s;
  // alarm off delay time - condition must clear for this long before being considered "gone"
  gr_AI_DP_CFFilter_Params.AlmLoOffDlyTime := T#1s;
  gr_AI_DP_CFFilter_Params.AlmHiOffDlyTime := T#1s;

  // Tank low level switch params
  gr_DI_LSL_CFTank_Params.Enable := FALSE; // H: process, L: Ignore. Not fitted. Set once fitted to enable processing and alarming
  gr_DI_LSL_CFTank_Params.AlmEnable := FALSE;
  // Sensor should be fail safe, so low signal is a low (alarm) level,
  gr_DI_LSL_CFTank_Params.AlmLoEnable := TRUE; // set to enable alarm if value is low
  gr_DI_LSL_CFTank_Params.AlmHiEnable := FALSE; // set to enable alarm if value is high
  gr_DI_LSL_CFTank_Params.Invert := FALSE;
  gr_DI_LSL_CFTank_Params.OnDlyTime := T#500ms; // delay time for value turning on
  gr_DI_LSL_CFTank_Params.OffDlyTime := T#500ms; // delay time for value turning off
  gr_DI_LSL_CFTank_Params.AlmLoOnDlyTime := T#3s;
  gr_DI_LSL_CFTank_Params.AlmHiOnDlyTime := T#1s;
  gr_DI_LSL_CFTank_Params.AlmLoOffDlyTime := T#1s;
  gr_DI_LSL_CFTank_Params.AlmHiOffDlyTime := T#1s;

  // Tank locator params
  gr_DI_ZS_CFTankLocator_Params.Enable := TRUE; // H: process, L: Ignore.
  gr_DI_ZS_CFTankLocator_Params.AlmEnable := TRUE;
  // Sensor should be fail safe, so low signal is an alarm
  gr_DI_ZS_CFTankLocator_Params.AlmLoEnable := TRUE; // set to enable alarm if value is low
  gr_DI_ZS_CFTankLocator_Params.AlmHiEnable := FALSE; // set to enable alarm if value is high
  gr_DI_ZS_CFTankLocator_Params.Invert := FALSE;
  gr_DI_ZS_CFTankLocator_Params.OnDlyTime := T#500ms; // delay time for value turning on
  gr_DI_ZS_CFTankLocator_Params.OffDlyTime := T#500ms; // delay time for value turning off
  gr_DI_ZS_CFTankLocator_Params.AlmLoOnDlyTime := T#3s;
  gr_DI_ZS_CFTankLocator_Params.AlmHiOnDlyTime := T#1s;
  gr_DI_ZS_CFTankLocator_Params.AlmLoOffDlyTime := T#1s;
  gr_DI_ZS_CFTankLocator_Params.AlmHiOffDlyTime := T#1s;

  // 480 VAC Monitor
  gr_DI_JI_480VACOk_Params.Enable := TRUE; // H: process, L: Ignore.
  // Indication only, no alarming needed.
  gr_DI_JI_480VACOk_Params.AlmEnable := FALSE;
  // Sensor should be fail safe, so low signal is an alarm
  gr_DI_JI_480VACOk_Params.AlmLoEnable := FALSE; // set to enable alarm if value is low
  gr_DI_JI_480VACOk_Params.AlmHiEnable := FALSE; // set to enable alarm if value is high
  gr_DI_JI_480VACOk_Params.Invert := FALSE;
  gr_DI_JI_480VACOk_Params.OnDlyTime := T#2s; // delay to make sure signal is present
  gr_DI_JI_480VACOk_Params.OffDlyTime := T#0ms; // delay time for value turning off
  gr_DI_JI_480VACOk_Params.AlmLoOnDlyTime := T#3s;
  gr_DI_JI_480VACOk_Params.AlmHiOnDlyTime := T#1s;
  gr_DI_JI_480VACOk_Params.AlmLoOffDlyTime := T#1s;
  gr_DI_JI_480VACOk_Params.AlmHiOffDlyTime := T#1s;

END_ACTION
```

### Program Logical/PlcLogic/Pendant (IEC)

#### fbEnabledAxis.sfc
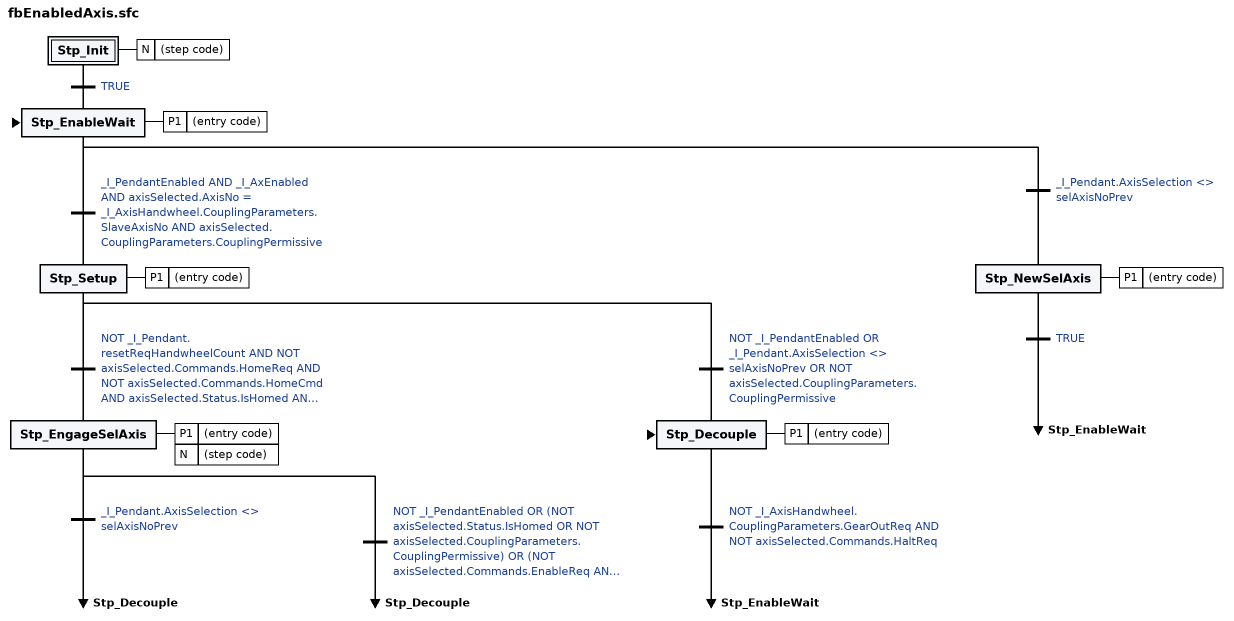
```iecst
FUNCTION_BLOCK fbEnabledAxis
INITIAL_STEP Stp_Init:
// Set current step (debugging purposes)
currentStep := STP_INIT;

// Pointers in sfc that are used in transitions
// may be dereferenced before execution begins ...
// so they need to point to something.
// Might as well pick the pointer passed in
axisSelected ACCESS _I_pAxisSelected;

// Set the previous axis selection so as to force an update
selAxisNoPrev := INVALID_SENTINEL;
END_STEP
TRANSITION FROM Stp_Init TO Stp_EnableWait:=
TRUE
END_TRANSITION
STEP Stp_EnableWait:
END_STEP
ENTRY_ACTION
// Set current step (debugging purposes)
currentStep := STP_ENABLE_WAIT;

// Get a snapshot of the axis selection so changes while processing are ignored, or at least
// handled at a time our our chosing.
// A pointer is used for access to prevent unnecessary copying of an axis structure (large)
// when 1) only a few elements are needed, and 2) the selected, and therefore referenced axis
// can change at any time.
 axisSelected ACCESS _I_pAxisSelected;
END_ACTION
TRANSITION pendant and ax enabled FROM Stp_EnableWait TO Stp_Setup:=
// Get on with it once pendant and axis is enabled and the
// slave axis matches the selected axis, and the slave axis is okay to couple
_I_PendantEnabled AND _I_AxEnabled AND
axisSelected.AxisNo = _I_AxisHandwheel.CouplingParameters.SlaveAxisNo AND
axisSelected.CouplingParameters.CouplingPermissive
END_TRANSITION
TRANSITION new axis is selected FROM Stp_EnableWait TO Stp_NewSelAxis:=
// New axis is selected
_I_Pendant.AxisSelection <> selAxisNoPrev
END_TRANSITION
STEP Stp_NewSelAxis:
END_STEP
ENTRY_ACTION
// Set current step
currentStep := STP_NEW_AXIS_SEL;

// Link selected axis to be a slave to the handwheel
_I_AxisHandwheel.CouplingParameters.SlaveAxisNo := axisSelected.AxisNo;
IF _I_AxisHandwheel.CouplingParameters.SlaveAxisNo = AD_SPINDLE THEN
  ;
  //_I_AxisHandwheel.SlaveAxisObj := gAxSpin;
ELSIF _I_AxisHandwheel.CouplingParameters.SlaveAxisNo = AD_SPINDLE THEN
;
END_IF;

END_ACTION
TRANSITION FROM Stp_NewSelAxis TO Stp_EnableWait:=
TRUE
END_TRANSITION
(* @SFCISJUMP := 'Stp_EnableWait' *)
STEP Stp_Setup:
END_STEP
ENTRY_ACTION
// Set current step (debugging purposes)
currentStep := STP_SETUP;

// Reset the handwheel counter. This
// guardes against rollover and allows
// starting from a predicted count.
_I_Pendant.resetReqHandwheelCount := TRUE;

// Home the virtual (handsheel) axis
// The virtual axis gets homed using direct mode
_I_AxisHandwheel.MoveParameters.HomeParams.Mode := mcHOMING_DIRECT;
_I_AxisHandwheel.MoveParameters.HomeParams.Position := 0.0;
_I_AxisHandwheel.Commands.HomeReq := TRUE;

// If the selected axis is not homed, request the axis be homed in position
IF NOT axisSelected.Status.IsHomed THEN
  axisSelected.MoveParameters.HomeParams.Mode := mcHOMING_DIRECT;
  axisSelected.MoveParameters.HomeParams.Position := axisSelected.Status.Position;
  axisSelected.Commands.HomeReq := TRUE;
END_IF;
END_ACTION
TRANSITION hw counter reset and axes homed FROM Stp_Setup TO Stp_EngageSelAxis:=
// Counter reset request should be handled (low) and
// the selected axis and handwheel axis should both be homed
NOT _I_Pendant.resetReqHandwheelCount AND
NOT axisSelected.Commands.HomeReq AND
NOT axisSelected.Commands.HomeCmd AND
axisSelected.Status.IsHomed AND
NOT _I_AxisHandwheel.Commands.HomeReq AND
NOT _I_AxisHandwheel.Commands.HomeCmd AND
_I_AxisHandwheel.Status.IsHomed AND
// The axis selection should still be the same
_I_Pendant.AxisSelection = selAxisNoPrev AND
// and the slave axis coupling permissive should still be good
axisSelected.CouplingParameters.CouplingPermissive
END_TRANSITION
TRANSITION pendant disabled or new axis seleted FROM Stp_Setup TO Stp_Decouple:=
// Pendant is disabled
NOT _I_PendantEnabled OR
// New axis is selected
_I_Pendant.AxisSelection <> selAxisNoPrev OR
// slave axis coupling permissive goes away
NOT axisSelected.CouplingParameters.CouplingPermissive

END_TRANSITION
STEP Stp_Decouple:
END_STEP
ENTRY_ACTION
// Set current step (debugging purposes)
currentStep := STP_DECOUPLE;

// Clear the gear in command, and halt the slave axis
_I_AxisHandwheel.CouplingParameters.GearOutReq := TRUE;
axisSelected.Commands.HaltReq := TRUE;
END_ACTION
TRANSITION decouple and halt req FROM Stp_Decouple TO Stp_EnableWait:=
// Make sure gear in command and halt req are clear, showing they've been at least seen
NOT _I_AxisHandwheel.CouplingParameters.GearOutReq AND
NOT axisSelected.Commands.HaltReq

END_TRANSITION
(* @SFCISJUMP := 'Stp_EnableWait' *)
STEP Stp_EngageSelAxis:
// Slave (selected axis) was geared in upon entry.

// Update the gear ratio if the speed selection changes
IF _I_Pendant.SpeedSelection <> selSpeedPrev THEN
  // update the snapshot to detect future changes
  selSpeedPrev := _I_Pendant.SpeedSelection;
  // Now update the gear ratio
  CalcGearRatioFb(_I_SlaveAxisDesignation := axisSelected.AxisNo, _I_SelectedSpeed := selSpeedPrev);
  _I_Pendant.GearRatioNumerator := CalcGearRatioFb._O_RatioNumerator;
  _I_Pendant.GearRatioDenominator := CalcGearRatioFb._O_RatioDenominator;
END_IF;
END_STEP
ENTRY_ACTION
// Set current step (debugging purposes)
currentStep := STP_ENGAGE_SEL_AX;

// At this point, both the handwheel and selected
// axis should be homed, and the selected axis should be enabled.
// The handwheel does not need to be (cannot be) enabled.
// Time to engage the selected axis as a slave.

// Snapshot the speed selection so changes can be detected
selSpeedPrev := _I_Pendant.SpeedSelection;

// Set the gear ratio based on the speed and axis selected
CalcGearRatioFb(_I_SlaveAxisDesignation := axisSelected.AxisNo,_I_SelectedSpeed := selSpeedPrev);
_I_Pendant.GearRatioNumerator := CalcGearRatioFb._O_RatioNumerator;
_I_Pendant.GearRatioDenominator := CalcGearRatioFb._O_RatioDenominator;

// Gear in the slave axis as long as the permissive is met
_I_AxisHandwheel.CouplingParameters.GearInReq := axisSelected.CouplingParameters.CouplingPermissive;
END_ACTION
TRANSITION new axis is selected FROM Stp_EngageSelAxis TO Stp_Decouple:=
// New axis is selected
_I_Pendant.AxisSelection <> selAxisNoPrev
END_TRANSITION
(* @SFCISJUMP := 'Stp_Decouple' *)
TRANSITION pendant or ax disabled FROM Stp_EngageSelAxis TO Stp_Decouple:=
// Pendant is disabled
NOT _I_PendantEnabled OR
// or the selected axis is no longer homed, or has lost coupling permissive, has lost the synchronized motion status
(NOT axisSelected.Status.IsHomed OR NOT axisSelected.CouplingParameters.CouplingPermissive) OR // OR axisSelected.Status.PlcOpenState <> mcAXIS_SYNCHRONIZED_MOTION) OR
// or selected axis is not enabled after request to do so has been processed -- this would usually be an alarm
(NOT axisSelected.Commands.EnableReq AND NOT axisSelected.Status.IsPoweredOn)
END_TRANSITION
(* @SFCISJUMP := 'Stp_Decouple' *)
END_FUNCTION_BLOCK
```

#### LocalFunctions.st
```iecst
// Decode 4 graycode inputs and return an axis designation
FUNCTION fctDecodeAxis
  (* A  B  C  D   Val   SwPos   Axis
     0  0  0  0   0     1 (X)   AD_X
     1  0  0  0   1     2 (Y)   AD_Y
     1  1  0  0   3     3 (Z)   AD_Z
     0  1  0  0   2     4 (4)   AD_OUTER_ECCENTRIC
     0  1  1  0   6     5 (5)   AD_INNER_ECCENTRIC
     1  1  1  0   7     6 (6)   AD_SPINDLE
      any other                 AD_UNKNOWN *)
  // Note D is always zero so that input param has a default of 0 (false)
  // Bit pack the values into an internal value to make value comparisons easier than
  // using each of the 4 inputs.
  // First init the value
  val := 0;
  val.0 := _InA;
  val.1 := _InB;
  val.2 := _InC;
  val.3 := _InD;
  IF val = 0 THEN
    fctDecodeAxis := AD_X;
  ELSIF val = 1 THEN
    fctDecodeAxis := AD_Y;
  ELSIF val = 3 THEN
    fctDecodeAxis := AD_Z;
  ELSIF val = 2 THEN
    fctDecodeAxis := AD_OUTER_ECCENTRIC;
  ELSIF val = 6 THEN
    fctDecodeAxis := AD_INNER_ECCENTRIC;
  ELSIF val = 7 THEN
    fctDecodeAxis := AD_SPINDLE;
  ELSE
    fctDecodeAxis := AD_UNKNOWN;
  END_IF;

END_FUNCTION

// Decode 4 graycode inputs and return a speed value
FUNCTION fctDecodeSpeed
  (* A  B  C  D   Val   Speed (Rtn value)
     0  0  0  0   0     0.0
     1  0  0  0   1     1.0
     1  1  0  0   3     10.0
     0  1  0  0   2     100.0
     0  1  1  0   6     1000.0
      any other         0         *)
  // Note D is always zero so that input param has a default of 0 (false)
  // Bit pack the values into an internal value to make value comparisons easier than
  // using each of the 4 inputs.
  // First init the value
  val := 0;
  val.0 := _InA;
  val.1 := _InB;
  val.2 := _InC;
  val.3 := _InD;
  IF val = 0 THEN
    fctDecodeSpeed := 0.0;
  ELSIF val = 1 THEN
    fctDecodeSpeed := 1.0;
  ELSIF val = 3 THEN
    fctDecodeSpeed := 10.0;
  ELSIF val = 2 THEN
    fctDecodeSpeed := 100.0;
  ELSIF val = 6 THEN
    fctDecodeSpeed := 1000.0;
  ELSE
    fctDecodeSpeed := 0.0;
  END_IF;

END_FUNCTION

FUNCTION_BLOCK fbCalcGearRatio (* Calc the selected axis:handwheel gear ratio *)
  (* Calc the gear ratio needed based on the selected slave, the selected speed
  and the measurement ratios.
  The handwheel has 100 indexed positions per turn.

  For the Z and X (depth) axes, the speed selections
  correspons to the following physical units per discrete handwheel index:
  Speed Select Value    HW Increment (in)   HW Increment (mm)   degrees
  0                     0                   0
  1.0                   0.0001              0.00254              0.0036
  10.0                  0.0010              0.0254               0.036
  100 .0                0.0100              0.254                0.36
  1000.0                0.1000              2.540                3.6 (360 degrees / 100 hw incr.)

  The ratio is calculated as follows:
  Numerator: Gear factor of the slave / Measurement resolution of the slave
  Denominator: Gear factor of the master / Measurement resolution of the master

  Spindle axis scaled 0-1 revolution,
  Outer and inner eccentrics scaled 0-360 degrees,
  Z scaled in mm
  *)

  // It turns out the numerator and denominator are big in all cases.
  // Keep the math to show the thinking, but divide by 100 to make the numbers friendlier
  IF _I_SlaveAxisDesignation = AD_SPINDLE THEN
    // At 1000 speed, slave goes 1 rev for every 360 degrees of the handwheel
    _O_RatioNumerator := REAL_TO_DINT(_I_SelectedSpeed * 1.0 / AXIS_SPINDLE_MEAS_RESOLUTION) / 100; // slave
    _O_RatioDenominator := REAL_TO_DINT(360.0 / AXIS_HW_MEAS_RESOLUTION) / 100; // master
  ELSIF _I_SlaveAxisDesignation = AD_OUTER_ECCENTRIC THEN
    // At 1000 speed, slave goes 360 for every 360 degrees of the handwheel
    _O_RatioNumerator := REAL_TO_DINT(_I_SelectedSpeed * 360.0 / AXIS_OUTE_MEAS_RESOLUTION) / 100; // slave
    _O_RatioDenominator := REAL_TO_DINT(360.0 / AXIS_HW_MEAS_RESOLUTION) / 100; // master
  ELSIF _I_SlaveAxisDesignation = AD_INNER_ECCENTRIC OR _I_SlaveAxisDesignation = AD_X THEN
    // Treat X and the inner eccentric the same
    // At 1000 speed, slave goes 360 for every 360 degrees of the handwheel
    _O_RatioNumerator := REAL_TO_DINT(_I_SelectedSpeed * 360.0 / AXIS_INE_MEAS_RESOLUTION) / 100; // slave
    _O_RatioDenominator := REAL_TO_DINT(360.0 / AXIS_HW_MEAS_RESOLUTION) / 100; // master
  ELSIF _I_SlaveAxisDesignation = AD_Z THEN
    // At 1000 speed, slave goes 0.1 * 100, or 10 inches (254 mm) for every 360 degrees of the handwheel
    (*
    _O_RatioNumerator := REAL_TO_DINT(_I_SelectedSpeed * 254.0 / AXIS_Z_MEAS_RESOLUTION) / 100; // slave
    _O_RatioDenominator := REAL_TO_DINT(360.0 / AXIS_HW_MEAS_RESOLUTION) / 100; // master
    *)
    // Test Values
    _O_RatioNumerator := 254; // slave
    _O_RatioDenominator := 3600; // master
  ELSE
    // Other axis
    // TODO: ? Error ? Use an arbitrary slow ratio
    _O_RatioNumerator := REAL_TO_DINT(_I_SelectedSpeed); // slave turns
    _O_RatioDenominator := REAL_TO_DINT(100.0); // master
  END_IF;

END_FUNCTION_BLOCK
```

### Program Logical/PlcLogic/CuttingFluidVFD (IEC)

#### Main.st - Init, cyclic, exit code
```iecst
PROGRAM _INIT

  // Flow established time
  timeCfFlowOk := T#5s;

END_PROGRAM

PROGRAM _CYCLIC

  // Process the alarms
  ProcessAlarms;

  cfVfd.isAllowedToStart :=
    (operatingMode.OperatingMode = OM_MANUAL_MODE OR
    operatingMode.OperatingMode = OM_PENDANT_MODE OR
    operatingMode.OperatingMode = OM_PRODUCTION_MODE) AND
    axes[AD_CF_VFD].Status.IsPoweredOn AND
    // VFD is present and waiting for next command, accel, or decel
    cfVfd.isModuleOk AND
    cfVfd.DevSpecStatus >= 2 AND
    cfVfd.DevSpecStatus <= 6 AND
    // axes[AD_CF_VFD].Status.IsHomed AND // homing not possible with inverter axis
    cfVfd.isLocated AND
    NOT cfVfd.isAlmLoLvlSw AND NOT cfVfd.isAlmLoFluid;

  cfVfd.isAllowedToRun :=
    cfVfd.isAllowedToStart AND
    NOT cfVfd.isAlmLoFlow AND
    NOT cfVfd.isAlmHiOutletPressure;
    // no device errors
    // cfVfd.DevSpecError = 0 AND
    // cfVfd.StdError = 0;

  // Map the axis status to the cf structure to get a running bit
  cfVfd.isRunning := axes[AD_CF_VFD].Status.IsMoveActive;

  // Determine when good flow is established -- time delay no flow problems
  tmrCfFlowOk(IN:= cfVfd.isRunning AND NOT cfVfd.isAlmLoFlow AND NOT cfVfd.isAlmLoOutletPressure, PT:= timeCfFlowOk);
  cfVfd.isFlowEstablished := tmrCfFlowOk.Q;

  // TESTING: Bypass CfVfd permits
  // cfVfd.isAllowedToStart := TRUE;
  // cfVfd.isAllowedToRun := TRUE;
  // cfVfd.isFlowEstablished := TRUE;
  // cfVfd.isRunning := TRUE;

END_PROGRAM

PROGRAM _EXIT
	(* Insert code here *)

END_PROGRAM
```

#### Action.st
```iecst
ACTION ProcessAlarms :
  // Alarm Enable/disable. These are permanent, but include here to easily make them dynamic.
  // Tank level
  gr_AI_LT_CFTankLevel_Params.AlmEnable := FALSE; // not fitted.
  // Flow
  gr_AI_FT_CFFlow_Params.AlmEnable := FALSE; // not fitted
  // Level switch
  gr_DI_LSL_CFTank_Params.AlmEnable := FALSE; // not fitted
  // Locator
  gr_DI_ZS_CFTankLocator_Params.AlmEnable:= TRUE;

  // Pressure and flow sensors -- enable while pump is running
  gr_AI_PT_CFPumpOutlet_Params.AlmEnable := cfVfd.isRunning;
  gr_AI_PT_CFFilterOutlet_Params.AlmEnable := FALSE; // cfVfd.isRunning; Don't an alarm on both HP gauges
  gr_AI_DP_CFFilter_Params.AlmEnable := cfVfd.isRunning;
  gr_AI_FT_CFFlow_Params.AlmEnable := cfVfd.isRunning;

  // Put alarm status into structure
  // isLocated
  cfVfd.isLocated := DI_ZS_CFTankLocator.alms = GAPIO_ALARM_NONE;

  // Level switch
  cfVfd.isAlmLoLvlSw := DI_LSL_CFTank.alms <> GAPIO_ALARM_NONE;

  // Flow
  // consider alarm on range, channel or lo lo alms
  almMask := 	GAPIO_ALARM_RANGEHI OR GAPIO_ALARM_RANGELO OR GAPIO_ALARM_CHANNEL OR GAPIO_ALARM_LOLO;
  cfVfd.isAlmLoFlow := (AI_FT_CFFlow.alms AND almMask) <> 0;
  // consider warning on lo alm
  almMask := GAPIO_ALARM_LO;
  cfVfd.isWarnLoFlow := (AI_FT_CFFlow.alms AND almMask) <> 0;

  // Fluid Level
  // consider alarm on range, channel or lo lo alms
  almMask := 	GAPIO_ALARM_RANGEHI OR GAPIO_ALARM_RANGELO OR GAPIO_ALARM_CHANNEL OR GAPIO_ALARM_LOLO;
  cfVfd.isAlmLoFluid := (AI_LT_CFTankLevel.alms AND almMask) <> 0;
  // consider warning on lo alm
  almMask := 	GAPIO_ALARM_LO;
  cfVfd.isWarnLoFluid := (AI_LT_CFTankLevel.alms AND almMask) <> 0;

  // Pump Outlet pressure
  // consider alarm on hi range, channel or hi hi alms
  almMask := 	GAPIO_ALARM_RANGEHI OR GAPIO_ALARM_CHANNEL OR GAPIO_ALARM_HIHI;
  cfVfd.isAlmHiOutletPressure := (AI_PT_CFPumpOutlet.alms AND almMask) <> 0;
  // consider alarm on range, channel or lo lo alms
  almMask := 	GAPIO_ALARM_RANGELO OR GAPIO_ALARM_LOLO;
  cfVfd.isAlmLoOutletPressure := (AI_PT_CFPumpOutlet.alms AND almMask) <> 0;
  // consider warning on lo alm
  almMask := 	GAPIO_ALARM_LO;
  cfVfd.isWarnLoOutletPressure := (AI_PT_CFPumpOutlet.alms AND almMask) <> 0;
  // consider warning on hi alm
  almMask := 	GAPIO_ALARM_HI;
  cfVfd.isWarnHiOutletPressure := (AI_PT_CFPumpOutlet.alms AND almMask) <> 0;

  // Hi Filter DP -- channel and range will trigger hi and low
  almMask := 	GAPIO_ALARM_RANGEHI OR GAPIO_ALARM_RANGELO OR GAPIO_ALARM_CHANNEL OR GAPIO_ALARM_HI;
  cfVfd.isWarnHiFilterDp := (AI_DP_CFFilter.alms AND almMask) <> 0;
  // Lo Filter DP -- channel and range will trigger hi and low
  almMask := 	GAPIO_ALARM_RANGEHI OR GAPIO_ALARM_RANGELO OR GAPIO_ALARM_CHANNEL OR GAPIO_ALARM_LO;
  cfVfd.isWarnLoFilterDp := (AI_DP_CFFilter.alms AND almMask) <> 0;

  // Alarm and warning summaries
  cfVfd.isWarnSummary := cfVfd.isWarnLoFlow OR cfVfd.isWarnLoFluid OR
  cfVfd.isWarnLoOutletPressure OR cfVfd.isWarnHiOutletPressure OR
  cfVfd.isWarnLoFilterDp OR cfVfd.isWarnHiFilterDp;

  cfVfd.isAlmSummary := cfVfd.isAlmLoFlow OR cfVfd.isAlmLoLvlSw OR
  cfVfd.isAlmLoFluid OR cfVfd.isAlmLoOutletPressure OR cfVfd.isAlmHiOutletPressure;

END_ACTION
```

### Program Logical/PlcLogic/OmSafeDev (IEC) - Operating Mode State Machine

#### OmSafeDev.typ
```iecst
TYPE
  (* Machine specific HMI axis requests. Intended to have one of these structures per axis. *)
  sHmiAxisReqs : STRUCT
    (* Boolean requests in this section. *)
    (* (none *)
    (* numerical requests *)
    (* (none *)
    (* hmi move type and direction selection related *)
    absMoveEnable : BOOL := TRUE; (* allow move type selection by default *)
    relMoveEnable : BOOL := TRUE;
    velMoveEnable : BOOL := TRUE;
    directionPosEnable : BOOL := TRUE; (* allow direction selection by default *)
    directionNegEnable : BOOL := TRUE;
    directionShortestEnable : BOOL := TRUE;
    moveDistanceEnable : BOOL := TRUE; (* enable params by default *)
    movePositionEnable : BOOL := TRUE;
    shiftEnable : BOOL := FALSE; (* coordinated axis shift enabled *)
    moveDesignation: DINT := -1; (* per hmi. 0: Abs, 1: Rel, 2:Vel or Jog, -1 is no selection. See fctDecodeHmiMoveType *)
    direction: DINT := -1; (* per hmi. 0: pos, 1: neg, 2: shortest, -1 is no selection. See fctDecodeHmiDirection *)
    (* axis designation. Two different data types for convenience. *)
    axisNo : USINT := 0; (* default to initial so setting a value can be detected. USINT for easy use in loops *)
    axisDesignation : eAXIS_DESIGNATION := AD_UNKNOWN; (* default to initial so setting a value can be detected *)
  END_STRUCT;

  (* Machine specific HMI process requests. Intended to have one of these per machine or otherwise as needed, but not per axis. *)
  sHmiProcessReqs : STRUCT
    (* Boolean requests in this section. *)
    (* NOTE/CAUTION These request bits may get cleared/copied by memcpy/memclr
    So be careful about adding boolean requests outside of this section.
    See ClearManualReqs action for example, in OmSaveDev program.
    Bool requests above zReqMoveUpLimit won't get auto cleared *)
    zReqMoveUpLimit : BOOL := FALSE;
    zReqMoveDownLimit : BOOL := FALSE;
    zReqMoveLUnL : BOOL := FALSE;
    zReqMoveSoc : BOOL := FALSE;
    zReqMoveIndexUp : BOOL := FALSE;
    zReqMoveIndexDown : BOOL := FALSE;
    zReqPosSocUseCurrent : BOOL := FALSE; (* set SOC to use the current position *)
    zReqPosSocUseSpecified :  BOOL := FALSE; (* set SOC to use the specified position *)
    zReqPosLUnLUseCurrent : BOOL := FALSE; (* set load/unload to use the current position *)
    zReqPosLUnLUseSpecified :  BOOL := FALSE; (* set load/unload to use the specified position *)
    cuttingHeadMoveReqRetract : BOOL := FALSE;
    (* NOTE/CAUTION Bool requests below cuttingHeadMoveReqRetract won't get auto cleared *)
    zMoveUpReqEnable : BOOL := FALSE; (* enable hmi request PBs *)
    zMoveDownReqEnable : BOOL := FALSE; (* enable hmi request PBs *)
    zMoveToSocReqEnable : BOOL := FALSE; (* enable hmi request PBs *)
    zMoveToLUnLReqEnable : BOOL := FALSE; (* enable hmi request PBs *)
    (* numerical values used with requests *)
    cuttingHeadReqDepth : LREAL := 0.0;
    zReqPosSoc : LREAL;
    zReqPosLUnL : LREAL;
  END_STRUCT;

END_TYPE
```

#### OmSafeDev.var
```iecst
VAR CONSTANT

END_VAR

VAR

  (* info from safety controller *)
  fs_AllSMsOk : BOOL;
  fs_EmoCmd : BOOL; (* H:Ok, L:EMO *)
  fs_EmoOwsActive : BOOL; (* H:Ok, L: EMO *)
  fs_EmoOwsOk : BOOL; (* H:Wiring Ok, L:Error *)
  fs_InSafeMode : BOOL; (* H:InSafeMode, L: Not in safe mode *)
  fs_KeyswitchInRun : BOOL; (* H:Run Pos, L: Not in run pos *)
  fs_KeyswitchOk : BOOL; (* H:Wiring Ok, L:Error *)
  fs_StartPbActive : BOOL; (* H:Start Req, L: Not pressed *)
  fs_StartPbOk : BOOL; (* H:Wiring Ok, L:Error *)
  fs_StopPbActive : BOOL; (* H: Allow Run, L: Stop *)
  fs_StopPbOk : BOOL; (* H:Wiring Ok, L:Error *)
  fs_CfGateClosed : BOOL; (* H:Closed, L: Open *)
  fs_CfGateClosedLocked : BOOL; (* H:Closed and locked(Ok), L: Open and/or unlocked *)
  fs_CfGateClosedOk : BOOL; (* H:Wiring Ok, L: Error *)

  (* info to safety controller *)
  ts_ResetEStop : BOOL;
  ts_ResetSafeMC : BOOL;
  ts_InEmoMode : BOOL;
  ts_InSafeMode : BOOL;
  ts_InPendantMode : BOOL;
  ts_InManualMode : BOOL;
  ts_InProductionMode : BOOL;

  (* cycle start/stop req *)
  tmrReqStartPulse : TP;
  tmrReqStopPulse : TP;

  (* EMO Reset *)
  timeEStopResetAllow : TIME;
  eStopResetAllowSecRemain : DINT;
  tmrEStopResetAllow : TON;
  timeResetPulse : TIME;
  tmrResetPulse : TP;

  (* HMI machine specific and axis requests *)
  hmiMachineAxisReqs : ARRAY[0..AXIS_COUNT] OF sHmiAxisReqs; (* machine specific requests that get turned into library reqs *)
  hmiLibraryAxisReqs : ARRAY[0..AXIS_COUNT] OF sMot_HmiAxisReqs; (* standard/basic requests handled by the library *)

  (* pointers used for memcpy/memset *)
  pSrc :  UDINT;
  pDest :  UDINT;
  byteCount :  UDINT;
  nxtAddr :  UDINT;

  (* axis index *)
  axisNo : DINT;

  (* fb to process Reqs *)
  procHmiProcessReqs : fbHandleHmiProcessReqs;
  procManualAxisReqsSpindle : fbHandleHmiAxisReq;
  procManualAxisReqsOutE : fbHandleHmiAxisReq;
  procManualAxisReqsInE : fbHandleHmiAxisReq;
  procManualAxisReqsZ : fbHandleHmiAxisReq;
  procManualAxisReqsHw : fbHandleHmiAxisReq;
  procManualAxisReqsCfVfd : fbHandleHmiAxisReq;
END_VAR
```

#### LocalFunctions.fun
```iecst
(* This function block will turn machine specific requests into GaMpMotion library requests,
and the library requests will handled with the motion library.
In this way, there is a cascading mechanism to get machine specific then axis
specific reqeusts processed by standard library functions,
even when process or machine specific things are not known by the library functions.
Note that the HMI binds to value in library axis req (sMot_HmiAxisReqs) for the move
requests, and move params. When controlling an individual axis, these are not machine specific.
This fb handles things like enable/disable choices based on selection, or other machine specific things. *)
FUNCTION_BLOCK fbHandleHmiAxisReq (* Turn machine specific reqs into GaMpMotion library requs, and then call library fb fbProcessHmiAxisReq. *)
  VAR_INPUT
    _I_MachineAxisReqs : REFERENCE TO sHmiAxisReqs;
    _I_LibraryAxisReqs : REFERENCE TO sMot_HmiAxisReqs;
    _I_Axis : REFERENCE TO sMot_Axis;
    _I_SlaveAxis : REFERENCE TO sMot_Axis;
    _I_AxisPositionLimits : REFERENCE TO sMot_PositionLimits;
  END_VAR

  VAR
    procLibraryReq : fbProcessHmiAxisReq; (* library function block to handle standard reqs built into library *)
  END_VAR
END_FUNCTION_BLOCK

(* This function block will turn process requests into GaMpMotion library requests.
The GA Motion Library requests will then be handled by the library.
In this way, there is a cascading mechanism to get process specific
reqeusts processed by standard library functions, even when process specific things
are not known by the library functions.*)
FUNCTION_BLOCK fbHandleHmiProcessReqs (* Turn process specific requests into GaMpMotion library requests. *)
  VAR_INPUT
    _I_ProcessReqs : REFERENCE TO sHmiProcessReqs;
    _I_WpCfg : REFERENCE TO sWp_Configuration;
    _I_pLibraryAxesReqs : UDINT; (* pointer to the beginning of the sMot_HmiAxisReqs [] *)
    _I_pAxis : UDINT; (* pointer to the beginning of the sMot_Axis [] *)
    _I_pAxisPositionLimits : UDINT; (* pointer to the beginning of the sMot_PositionLimits [] *)
  END_VAR

  VAR
    (* These references are used to call the procLibraryReq function.
    They are set by logic to specific array members by calculating an
    offset from the pointers passed in *)
    rLibReqs : REFERENCE TO sMot_HmiAxisReqs;
    rAxis : REFERENCE TO sMot_Axis;
    rSlaveAxis : REFERENCE TO sMot_Axis;
    rAxisPositionLimits : REFERENCE TO sMot_PositionLimits;
    slaveNum : USINT; (* hold looked up slave number *)
    (* calc sizes for convenience *)
    szLibReq : UDINT;
    szAxis : UDINT;
    szAxisPosLimits : UDINT;
    procLibraryReq : fbProcessHmiAxisReq; (* library function block to handle standard reqs built into library *)
    (* for use with brsmemset *)
    pSrc : UDINT;
    pDest : UDINT;
    byteCount : UDINT;
    nextAddr : UDINT;
  END_VAR
END_FUNCTION_BLOCK

(* The HMI can easily set values like 0, 1, 2 from radio buttons, but it is harder to set specific move type values *)
(* This function is intended to take an HMI selection and return a direction usable by the McAxis library *)
FUNCTION fctDecodeHmiDirection : McDirectionEnum (* Take in an HMI move type and return a corresponding enum move designation *)
  VAR_INPUT
    _I_DirectionReq : DINT;
  END_VAR
END_FUNCTION

(* The HMI can easily set values like 0, 1, 2 from radio buttons, but it is harder to set specific move type values *)
(* This function is intended to take an HMI selection and return a move type usable by the GaMpMotion library *)
FUNCTION fctDecodeHmiMoveType : eGAMOT_MOVE_DESIGNATION (* Take in an HMI move type and return a corresponding enum move designation *)
  VAR_INPUT
    _I_AxisIsEndless : BOOL;
    _I_MoveReq : DINT;
    _I_MoveDirection : McDirectionEnum;
  END_VAR
END_FUNCTION

(* The HMI can easily set values like 0, 1, 2 from radio buttons, but it is harder to set specific sub mode values. *)
(* This function is intended to take an HMI selection and return a sub mode usable by the PLC logic. *)
FUNCTION fctDecodeHmiSubMode : WORD (* Take in an HMI sub mode selection and return a corresponding sub mode *)
  VAR_INPUT
    _I_SubModeReq : SINT;
  END_VAR
END_FUNCTION
```

#### Action.st
```iecst
ACTION ClearProcessReqs :
  // Clear Process Reqs, and then the machine specific axis Reqs
  // Process Reqs
  // Bool reqs
  pSrc := ADR(hmiProcessReqs.StartOfClearedRequests);
  pDest := ADR(hmiProcessReqs.EndOfClearedRequests);
  byteCount := pDest - pSrc + SIZEOF(BOOL);
  nxtAddr := brsmemset(pSrc, 0, byteCount);
END_ACTION

ACTION ClearMotionReqs :
  // Clear Process Reqs, and then the machine specific axis Reqs
  // Process Reqs
  // Bool reqs
  pSrc := ADR(hmiProcessReqs.StartOfClearedRequests);
  pDest := ADR(hmiProcessReqs.EndOfClearedRequests);
  byteCount := pDest - pSrc + SIZEOF(BOOL);
  nxtAddr := brsmemset(pSrc, 0, byteCount);

  // Now clear the machine specific axis reqs
  FOR axisNo := 0 TO AXIS_COUNT DO
    // Bool reqs
    // (none)
    // numerical requests
    // (none)
    // move type and direction
    hmiMachineAxisReqs[axisNo].moveDesignation := -1; (* clear HMI selection *)
    hmiMachineAxisReqs[axisNo].direction := -1; (* clear HMI selection *)

    // Now clear the library requests
    // Bool reqs
    pSrc := ADR(hmiLibraryAxisReqs[axisNo].moveReq);
    pDest := ADR(hmiLibraryAxisReqs[axisNo].disengageSlaveReq);
    byteCount := pDest - pSrc + SIZEOF(BOOL);
    nxtAddr := brsmemset(pSrc, 0, byteCount);
    // numerical requests
    hmiLibraryAxisReqs[axisNo].Position := 0.0;
    hmiLibraryAxisReqs[axisNo].Distance := 0.0;
    hmiLibraryAxisReqs[axisNo].Velocity := 0.0;
    // move type and direction
    hmiLibraryAxisReqs[axisNo].moveDesignation := GAMOT_MD_NO_MOVE_COMMANDED;
    hmiLibraryAxisReqs[axisNo].Direction := mcDIR_UNDEFINED;
  END_FOR;

END_ACTION

ACTION ClearNonMotionReqs :
  // Clear the non-motion reqs
  FOR axisNo := 0 TO AXIS_COUNT DO
    // Clear requests to set limits and requests to reset
    // Bool reqs
    pSrc := ADR(hmiLibraryAxisReqs[axisNo].setPositionLimitsReq);
    pDest := ADR(hmiLibraryAxisReqs[axisNo].driveResetReq);
    byteCount := pDest - pSrc + SIZEOF(BOOL);
    nxtAddr := brsmemset(pSrc, 0, byteCount);
    // numerical requests
    // (none)
  END_FOR;

END_ACTION

ACTION ClearCycleReqs :
  // TODO: Does Cycle start/stop have a meaning in manual mode?
  // For now block them
  operatingMode.ReqCycleStart := FALSE;
  operatingMode.ReqCycleStop := FALSE;
  operatingMode.HmiReqCycleStart := FALSE;
  operatingMode.HmiReqCycleStop:= FALSE;
  operatingMode.ReqEmoReset := FALSE;
END_ACTION

ACTION ManualModeAxisPermits :
  // In Manual Mode
  // cycle is not okay to run
  cyclePermissives.isOmOk := FALSE;

  // TODO: Proper permissions. For now, wide open
  axes[AD_SPINDLE].MoveParameters.PosMovePermissive := TRUE;
  axes[AD_SPINDLE].MoveParameters.NegMovePermissive := TRUE;

  axes[AD_OUTER_ECCENTRIC].MoveParameters.PosMovePermissive := TRUE;
  axes[AD_OUTER_ECCENTRIC].MoveParameters.NegMovePermissive := TRUE;

  axes[AD_INNER_ECCENTRIC].MoveParameters.PosMovePermissive := TRUE;
  axes[AD_INNER_ECCENTRIC].MoveParameters.NegMovePermissive := TRUE;

  axes[AD_Z].MoveParameters.PosMovePermissive := TRUE;
  axes[AD_Z].MoveParameters.NegMovePermissive := TRUE;

  // Handwheel is virtual -- don't allow moves
  axes[AD_HANDWHEEL].MoveParameters.PosMovePermissive := FALSE;
  axes[AD_HANDWHEEL].MoveParameters.NegMovePermissive := FALSE;

  // cutting fluid pump
  axes[AD_CF_VFD].MoveParameters.PosMovePermissive := cfVfd.isAllowedToRun;
// Allow forward running only
  axes[AD_CF_VFD].MoveParameters.NegMovePermissive := FALSE;

END_ACTION

ACTION PendantModeAxisPermits :
    // In Pendant Mode
    // cycle is not okay to run
  cyclePermissives.isOmOk := FALSE;

  // TODO: Proper permissions. For now, wide open
  axes[AD_SPINDLE].MoveParameters.PosMovePermissive := TRUE;
  axes[AD_SPINDLE].MoveParameters.NegMovePermissive := TRUE;

  axes[AD_OUTER_ECCENTRIC].MoveParameters.PosMovePermissive := TRUE;
  axes[AD_OUTER_ECCENTRIC].MoveParameters.NegMovePermissive := TRUE;

  axes[AD_INNER_ECCENTRIC].MoveParameters.PosMovePermissive := TRUE;
  axes[AD_INNER_ECCENTRIC].MoveParameters.NegMovePermissive := TRUE;

  axes[AD_Z].MoveParameters.PosMovePermissive := TRUE;
  axes[AD_Z].MoveParameters.NegMovePermissive := TRUE;

  // Handwheel is virtual -- don't allow moves
  axes[AD_HANDWHEEL].MoveParameters.PosMovePermissive := FALSE;
  axes[AD_HANDWHEEL].MoveParameters.NegMovePermissive := FALSE;

  // cutting fluid pump
  axes[AD_CF_VFD].MoveParameters.PosMovePermissive := cfVfd.isAllowedToRun;
// Allow forward running only
  axes[AD_CF_VFD].MoveParameters.NegMovePermissive := FALSE;

END_ACTION

ACTION ProductionModeAxisPermits :
  // In Production Mode
  // cycle is okay to run
  cyclePermissives.isOmOk := TRUE;

  // Spindle
  // TODO: mask requests or commands?
  // fctClearMotionRequests(_I_ReqMask := MACM_NOMASK, _IO_Commands := axes[AD_SPINDLE].Commands);
  // Spindle is allowed to move forward as long as the cutting fluid is running
  // Spindle cannot run backward
  axes[AD_SPINDLE].MoveParameters.PosMovePermissive := cfVfd.isRunning AND cfVfd.isFlowEstablished;
  axes[AD_SPINDLE].MoveParameters.NegMovePermissive := FALSE;

  // Outer Eccentric
  // TODO: mask requests or commands?
  // fctClearMotionRequests(_I_ReqMask := MACM_NOMASK, _IO_Commands := axes[AD_OUTER_ECCENTRIC].Commands);
  // TODO: require spindle to be moving?
  axes[AD_OUTER_ECCENTRIC].MoveParameters.PosMovePermissive := TRUE;
  axes[AD_OUTER_ECCENTRIC].MoveParameters.NegMovePermissive := TRUE;
  // TODO: mask requests or commands?

  // Inner Eccentric
  // TODO: mask requests or commands?
  // fctClearMotionRequests(_I_ReqMask := MACM_NOMASK, _IO_Commands := axes[AD_INNER_ECCENTRIC].Commands);
  axes[AD_INNER_ECCENTRIC].MoveParameters.PosMovePermissive := TRUE;
  axes[AD_INNER_ECCENTRIC].MoveParameters.NegMovePermissive := TRUE;
  // TODO: mask requests or commands?

  // Z
  // Axis needs to homed and enabled, but also,
  // moving Z Axis requires the cutting head to be retracted.
  // Therefore the inner and outer both need to be homed, so the position is known,
  // and the difference in posiiton (axis.Status.CalculatedPosition1) needs to be within
  // tolerance.
  axes[AD_Z].MoveParameters.PosMovePermissive :=
    axes[AD_Z].Status.IsHomed AND axes[AD_Z].Status.IsPoweredOn AND
    axes[AD_INNER_ECCENTRIC].Status.IsHomed AND axes[AD_OUTER_ECCENTRIC].Status.IsHomed AND
    ABS(axes[AD_INNER_ECCENTRIC].Status.CalculatedPosition1) < TOL_DEPTH_ZERO_DEG AND
    // position must be less than limit
    axes[AD_Z].Status.Position <= gr_AxisPositionLimits[AD_Z].PositionLimitPos;

  axes[AD_Z].MoveParameters.NegMovePermissive :=
    axes[AD_Z].Status.IsHomed AND axes[AD_Z].Status.IsPoweredOn AND
    axes[AD_INNER_ECCENTRIC].Status.IsHomed AND axes[AD_OUTER_ECCENTRIC].Status.IsHomed AND
    ABS(axes[AD_INNER_ECCENTRIC].Status.CalculatedPosition1) < TOL_DEPTH_ZERO_DEG AND
    // position must be less than limit
    axes[AD_Z].Status.Position >= gr_AxisPositionLimits[AD_Z].PositionLimitNeg;

  // Set process related enable/disables
  hmiProcessReqs.zMoveDownReqEnable := axes[AD_Z].MoveParameters.NegMovePermissive;
  hmiProcessReqs.zMoveUpReqEnable := axes[AD_Z].MoveParameters.PosMovePermissive;
  hmiProcessReqs.zMoveToLUnLReqEnable :=
    // okay to go up
    (axes[AD_Z].Status.Position < gr_CfgCurrent.zAxis.loadUnloadPos AND axes[AD_Z].MoveParameters.PosMovePermissive) OR
    // okay to go down
    (axes[AD_Z].Status.Position > gr_CfgCurrent.zAxis.loadUnloadPos AND axes[AD_Z].MoveParameters.NegMovePermissive);
  hmiProcessReqs.zMoveToSocReqEnable :=
    // okay to go up
    (axes[AD_Z].Status.Position < gr_CfgCurrent.zAxis.startOfCutPos AND axes[AD_Z].MoveParameters.PosMovePermissive) OR
    // okay to go down
    (axes[AD_Z].Status.Position > gr_CfgCurrent.zAxis.startOfCutPos AND axes[AD_Z].MoveParameters.NegMovePermissive);

  // Handwheel is virtual -- don't allow moves
  axes[AD_HANDWHEEL].MoveParameters.PosMovePermissive := FALSE;
  axes[AD_HANDWHEEL].MoveParameters.NegMovePermissive := FALSE;

  // cutting fluid pump
  axes[AD_CF_VFD].MoveParameters.PosMovePermissive := cfVfd.isAllowedToRun;
  hmiProcessReqs.cfRunEnable := axes[AD_CF_VFD].MoveParameters.PosMovePermissive;
// Allow forward running only
  axes[AD_CF_VFD].MoveParameters.NegMovePermissive := FALSE;

END_ACTION

ACTION OtherModeAxisPermits:
    // Not in a mode (safe, initial, unknown, etc.)
    // This is some sort of error -- don't allow any motion
    // For each axis clear the requestes, and the move permissives
    // TODO: Clear the commnads?

    // cycle is no okay to run
  cyclePermissives.isOmOk := FALSE;

  // Spindle
  fctClearMotionRequests(_I_ReqMask := MACM_NOMASK, _IO_Commands := axes[AD_SPINDLE].Commands);
  // TODO: Clear the commnads, or let the axis SM handle it?
  // fctClearMotionCommands(_I_CmdMask := MACM_NOMASK, _IO_Commands := axes[AD_SPINDLE].Commands);
  axes[AD_SPINDLE].MoveParameters.PosMovePermissive := FALSE;
  axes[AD_SPINDLE].MoveParameters.NegMovePermissive := FALSE;

  // Outer Eccentric
  fctClearMotionRequests(_I_ReqMask := MACM_NOMASK, _IO_Commands := axes[AD_OUTER_ECCENTRIC].Commands);
  // TODO: Clear the commnads, or let the axis SM handle it?
  // fctClearMotionCommands(_I_CmdMask := MACM_NOMASK, _IO_Commands := axes[AD_OUTER_ECCENTRIC].Commands);
  axes[AD_OUTER_ECCENTRIC].MoveParameters.PosMovePermissive := FALSE;
  axes[AD_OUTER_ECCENTRIC].MoveParameters.NegMovePermissive := FALSE;

  // Inner Eccentric
  fctClearMotionRequests(_I_ReqMask := MACM_NOMASK, _IO_Commands := axes[AD_INNER_ECCENTRIC].Commands);
  // TODO: Clear the commnads, or let the axis SM handle it?
  // fctClearMotionCommands(_I_CmdMask := MACM_NOMASK, _IO_Commands := axes[AD_INNER_ECCENTRIC].Commands);
  axes[AD_INNER_ECCENTRIC].MoveParameters.PosMovePermissive := FALSE;
  axes[AD_INNER_ECCENTRIC].MoveParameters.NegMovePermissive := FALSE;

  // Z
  fctClearMotionRequests(_I_ReqMask := MACM_NOMASK, _IO_Commands := axes[AD_Z].Commands);
  // TODO: Clear the commnads, or let the axis SM handle it?
  // fctClearMotionCommands(_I_CmdMask := MACM_NOMASK, _IO_Commands := axes[AD_Z].Commands);
  axes[AD_Z].MoveParameters.PosMovePermissive := FALSE;
  axes[AD_Z].MoveParameters.NegMovePermissive := FALSE;

  // cutting fluid pump
  axes[AD_CF_VFD].MoveParameters.PosMovePermissive := cfVfd.isAllowedToRun;
// Allow forward running only
  axes[AD_CF_VFD].MoveParameters.NegMovePermissive := FALSE;

END_ACTION

ACTION ModeIndependentPermissions :
  // Set status and permissive related things that are independent of mode

  // Rollup of cycle start  allowed
  cyclePermissives.allowCycleStart :=
  // Operating mode must be okay
  cyclePermissives.isOmOk AND
  // Cutting fluid must be okay to start
  cfVfd.isAllowedToStart AND
    // Each axis needs to be in standstill or disabled. Additionally, inner eccentric can be coupled.
  (axes[AD_SPINDLE].Status.PlcOpenState = mcAXIS_DISABLED OR axes[AD_SPINDLE].Status.PlcOpenState = mcAXIS_STANDSTILL) AND
  (axes[AD_OUTER_ECCENTRIC].Status.PlcOpenState = mcAXIS_DISABLED OR axes[AD_OUTER_ECCENTRIC].Status.PlcOpenState = mcAXIS_STANDSTILL) AND
  (axes[AD_INNER_ECCENTRIC].Status.PlcOpenState = mcAXIS_DISABLED OR axes[AD_INNER_ECCENTRIC].Status.PlcOpenState = mcAXIS_STANDSTILL OR axes[AD_INNER_ECCENTRIC].Status.PlcOpenState = mcAXIS_SYNCHRONIZED_MOTION) AND
  (axes[AD_Z].Status.PlcOpenState = mcAXIS_DISABLED OR axes[AD_Z].Status.PlcOpenState = mcAXIS_STANDSTILL) AND
  // axes need to be referenced, and not force to be re-referenced
  axes[AD_SPINDLE].Status.IsHomed AND NOT axes[AD_SPINDLE].ForceSetRef AND
  axes[AD_OUTER_ECCENTRIC].Status.IsHomed AND NOT axes[AD_OUTER_ECCENTRIC].ForceSetRef AND
  axes[AD_INNER_ECCENTRIC].Status.IsHomed AND NOT axes[AD_INNER_ECCENTRIC].ForceSetRef AND
  axes[AD_Z].Status.IsHomed AND NOT axes[AD_Z].ForceSetRef AND
  // axes need to be calibrated to the process
  // Z will be indexed when the cycle is started, so no need to check it here, as long as Z is calibrated
  gr_PartCurrent.isZCalibrated AND gr_PartCurrent.isInECalibrated AND gr_PartCurrent.isOutECalibrated;

  // Rollup of cycle run allowed
  cyclePermissives.allowCycleRun :=
  // Operating mode must be okay
  cyclePermissives.isOmOk AND
  // Cutting fluid must be okay to start
  cfVfd.isAllowedToStart AND
    // Axes can't be in error or homing. Disabled is allowed because the cycle may start with them disabled.
  (axes[AD_SPINDLE].Status.PlcOpenState <> mcAXIS_ERRORSTOP AND axes[AD_SPINDLE].Status.PlcOpenState <> mcAXIS_HOMING) AND
  (axes[AD_OUTER_ECCENTRIC].Status.PlcOpenState <> mcAXIS_ERRORSTOP AND axes[AD_OUTER_ECCENTRIC].Status.PlcOpenState <> mcAXIS_HOMING) AND
  (axes[AD_INNER_ECCENTRIC].Status.PlcOpenState <> mcAXIS_ERRORSTOP AND axes[AD_INNER_ECCENTRIC].Status.PlcOpenState <> mcAXIS_HOMING) AND
  (axes[AD_Z].Status.PlcOpenState <> mcAXIS_ERRORSTOP AND axes[AD_Z].Status.PlcOpenState <> mcAXIS_HOMING) AND
  // axes need to be referenced, and not force to be re-referenced
  axes[AD_SPINDLE].Status.IsHomed AND NOT axes[AD_SPINDLE].ForceSetRef AND
  axes[AD_OUTER_ECCENTRIC].Status.IsHomed AND NOT axes[AD_OUTER_ECCENTRIC].ForceSetRef AND
  axes[AD_INNER_ECCENTRIC].Status.IsHomed AND NOT axes[AD_INNER_ECCENTRIC].ForceSetRef AND
  axes[AD_Z].Status.IsHomed AND NOT axes[AD_Z].ForceSetRef AND
  // axes need to be calibrated to the process
  // Z will be indexed when the cycle is started, so no need to check it here, as long as Z is calibrated
  gr_PartCurrent.isZCalibrated AND gr_PartCurrent.isInECalibrated AND gr_PartCurrent.isOutECalibrated;
END_ACTION
```
